// ---- DUTs/IO/PDOs/Channel_3263D8D5.TcDUT
{attribute 'GeneratedUsingTerminal: KL8524'}
{attribute addProperty BoxType "KL8524"}
{attribute addProperty Id "StateAT %I*USINT0Auto_Manual_ChannelAT %I*BYTE0Switch_modeAT %I*BYTE0On_Off_ChannelAT %I*BYTE0CtrlAT %Q*USINT0Switch_mode_OutAT %Q*BYTE0Data_Reg_ComAT %Q*BYTE0LED_Out_greenAT %Q*BYTE0LED_Out_yellowAT %Q*BYTE0"}
{attribute addProperty CRC "845404373"}
{attribute addProperty Size "0"}
TYPE Channel_3263D8D5 :
STRUCT
	{attribute addProperty Name "State"}
	State AT %I* : USINT;
	{attribute addProperty Name "Auto_Manual_Channel"}
	Auto_Manual_Channel AT %I* : BYTE;
	{attribute addProperty Name "Switch_mode"}
	Switch_mode AT %I* : BYTE;
	{attribute addProperty Name "On_Off_Channel"}
	On_Off_Channel AT %I* : BYTE;
	{attribute addProperty Name "Ctrl"}
	Ctrl AT %Q* : USINT;
	{attribute addProperty Name "Switch_mode_Out"}
	Switch_mode_Out AT %Q* : BYTE;
	{attribute addProperty Name "Data_Reg_Com"}
	Data_Reg_Com AT %Q* : BYTE;
	{attribute addProperty Name "LED_Out_green"}
	LED_Out_green AT %Q* : BYTE;
	{attribute addProperty Name "LED_Out_yellow"}
	LED_Out_yellow AT %Q* : BYTE;
END_STRUCT
END_TYPE

// ---- DUTs/IO/PDOs/Channel_D490E973.TcDUT
{attribute 'GeneratedUsingTerminal: KL8528'}
{attribute addProperty BoxType "KL8528"}
{attribute addProperty Id "StateAT %I*USINT0Auto_Manual_ChannelAT %I*BYTE0On_Off_ChannelAT %I*BYTE0CtrlAT %Q*USINT0OutAT %Q*BYTE0Data_Reg_ComAT %Q*BYTE0LED_Out_greenAT %Q*BYTE0LED_Out_yellowAT %Q*BYTE0"}
{attribute addProperty CRC "3566266739"}
{attribute addProperty Size "0"}
TYPE Channel_D490E973 :
STRUCT
	{attribute addProperty Name "State"}
	State AT %I* : USINT;
	{attribute addProperty Name "Auto_Manual_Channel"}
	Auto_Manual_Channel AT %I* : BYTE;
	{attribute addProperty Name "On_Off_Channel"}
	On_Off_Channel AT %I* : BYTE;
	{attribute addProperty Name "Ctrl"}
	Ctrl AT %Q* : USINT;
	{attribute addProperty Name "Out"}
	Out AT %Q* : BYTE;
	{attribute addProperty Name "Data_Reg_Com"}
	Data_Reg_Com AT %Q* : BYTE;
	{attribute addProperty Name "LED_Out_green"}
	LED_Out_green AT %Q* : BYTE;
	{attribute addProperty Name "LED_Out_yellow"}
	LED_Out_yellow AT %Q* : BYTE;
END_STRUCT
END_TYPE

// ---- DUTs/IO/PDOs/KL_6576A681.TcDUT
{attribute 'GeneratedUsingTerminal: KL8610'}
{attribute addProperty BoxType "KL8610"}
{attribute addProperty Id "StateAT %I*USINT0Data_InAT %I*INT0CtrlAT %Q*USINT0Data_OutAT %Q*INT0"}
{attribute addProperty CRC "1702274689"}
{attribute addProperty Size "0"}
TYPE KL_6576A681 :
STRUCT
	{attribute addProperty Name "State"}
	State AT %I* : USINT;
	{attribute addProperty Name "Data_In"}
	Data_In AT %I* : INT;
	{attribute addProperty Name "Ctrl"}
	Ctrl AT %Q* : USINT;
	{attribute addProperty Name "Data_Out"}
	Data_Out AT %Q* : INT;
END_STRUCT
END_TYPE

// ---- DUTs/IO/PDOs/Channel_64AAC8C7.TcDUT
{attribute 'GeneratedUsingTerminal: KL9110'}
{attribute addProperty BoxType "KL9110"}
{attribute addProperty Id "PowerAT %I*BOOL0ShortCircuitAT %I*BOOL0"}
{attribute addProperty CRC "1688914119"}
{attribute addProperty Size "0"}
TYPE Channel_64AAC8C7 EXTENDS InputBase_8311D824 :
STRUCT
	{attribute addProperty Name "Power"}
	Power AT %I* : BOOL;
	{attribute addProperty Name "ShortCircuit"}
	ShortCircuit AT %I* : BOOL;
END_STRUCT
END_TYPE

// ---- DUTs/IO/PDOs/Channel_471FAA5C.TcDUT
{attribute 'GeneratedUsingTerminal: KL9191'}
{attribute addProperty BoxType "KL9191"}
{attribute addProperty Id "Contact_DI1AT %I*BOOL0Contact_DI2AT %I*BOOL0Contact_DI3AT %I*BOOL0LED_DO1AT %Q*BOOL0Relay_2kWAT %Q*BOOL0Relay_FAN1AT %Q*BOOL0Relay_FAN2AT %Q*BOOL0Relay_FAN3AT %Q*BOOL0TRIAC_Y1AT %Q*BOOL0TRIAC_Y2AT %Q*BOOL0"}
{attribute addProperty CRC "1193257564"}
{attribute addProperty Size "0"}
TYPE Channel_471FAA5C :
STRUCT
	{attribute addProperty Name "Contact_DI1"}
	Contact_DI1 AT %I* : BOOL;
	{attribute addProperty Name "Contact_DI2"}
	Contact_DI2 AT %I* : BOOL;
	{attribute addProperty Name "Contact_DI3"}
	Contact_DI3 AT %I* : BOOL;
	{attribute addProperty Name "LED_DO1"}
	LED_DO1 AT %Q* : BOOL;
	{attribute addProperty Name "Relay_2kW"}
	Relay_2kW AT %Q* : BOOL;
	{attribute addProperty Name "Relay_FAN1"}
	Relay_FAN1 AT %Q* : BOOL;
	{attribute addProperty Name "Relay_FAN2"}
	Relay_FAN2 AT %Q* : BOOL;
	{attribute addProperty Name "Relay_FAN3"}
	Relay_FAN3 AT %Q* : BOOL;
	{attribute addProperty Name "TRIAC_Y1"}
	TRIAC_Y1 AT %Q* : BOOL;
	{attribute addProperty Name "TRIAC_Y2"}
	TRIAC_Y2 AT %Q* : BOOL;
END_STRUCT
END_TYPE

// ---- DUTs/IO/PDOs/Diag_1F4F4573.TcDUT
{attribute 'GeneratedUsingTerminal: KL9505-0010'}
{attribute addProperty BoxType "KL9505-0010"}
{attribute addProperty Id "Supply_Voltage_OKAT %I*BOOL0Over_currentAT %I*BOOL0"}
{attribute addProperty CRC "525288819"}
{attribute addProperty Size "0"}
TYPE Diag_1F4F4573 EXTENDS InputBase_8311D824 :
STRUCT
	{attribute addProperty Name "Supply_Voltage_OK"}
	Supply_Voltage_OK AT %I* : BOOL;
	{attribute addProperty Name "Over_current"}
	Over_current AT %I* : BOOL;
END_STRUCT
END_TYPE

// ---- DUTs/IO/PDOs/Channel_0029832E.TcDUT
{attribute 'GeneratedUsingTerminal: KL9528'}
{attribute addProperty BoxType "KL9528"}
{attribute addProperty Id "OverloadAT %I*BOOL0UndervoltageAT %I*BOOL0ResetAT %Q*BOOL0"}
{attribute addProperty CRC "2720558"}
{attribute addProperty Size "0"}
TYPE Channel_0029832E :
STRUCT
	{attribute addProperty Name "Overload"}
	Overload AT %I* : BOOL;
	{attribute addProperty Name "Undervoltage"}
	Undervoltage AT %I* : BOOL;
	{attribute addProperty Name "Reset"}
	Reset AT %Q* : BOOL;
END_STRUCT
END_TYPE

// ---- DUTs/IO/PDOs/Channel_12652743.TcDUT
{attribute 'GeneratedUsingTerminal: KL9999'}
{attribute addProperty BoxType "KL9999"}
{attribute addProperty Id "VarInAT %I*UINT0VarOutAT %Q*UINT0"}
{attribute addProperty CRC "308619075"}
{attribute addProperty Size "0"}
TYPE Channel_12652743 :
STRUCT
	{attribute addProperty Name "VarIn"}
	VarIn AT %I* : UINT;
	{attribute addProperty Name "VarOut"}
	VarOut AT %Q* : UINT;
END_STRUCT
END_TYPE

// ---- DUTs/IO/PDOs/InfoData_E68C61CD.TcDUT
{attribute 'GeneratedUsingTerminal: IODEVICETYPE_ETHERCATPROT'}
{attribute addProperty BoxType "IODEVICETYPE_ETHERCATPROT"}
{attribute addProperty Id "ChangeCountAT %I*UINT2DevIdAT %I*UINT2AmsNetIdAT %I*AMSNETID6CfgSlaveCountAT %I*UINT2DcToTcTimeOffsetAT %I*LINT8DcToExtTimeOffsetAT %I*LINT8"}
{attribute addProperty CRC "3867959757"}
{attribute addProperty Size "28"}
TYPE InfoData_E68C61CD EXTENDS InputBase_8311D824 :
STRUCT
	{attribute addProperty Name "ChangeCount"}
	ChangeCount AT %I* : UINT;
	{attribute addProperty Name "DevId"}
	DevId AT %I* : UINT;
	{attribute addProperty Name "AmsNetId"}
	AmsNetId AT %I* : AMSNETID;
	{attribute addProperty Name "CfgSlaveCount"}
	CfgSlaveCount AT %I* : UINT;
	{attribute addProperty Name "DcToTcTimeOffset"}
	DcToTcTimeOffset AT %I* : LINT;
	{attribute addProperty Name "DcToExtTimeOffset"}
	DcToExtTimeOffset AT %I* : LINT;
END_STRUCT
END_TYPE

// ---- DUTs/IO/PDOs/WcState_0B2B16F9.TcDUT
{attribute 'GeneratedUsingTerminal: IODEVICETYPE_ETHERCATPROT'}
{attribute addProperty BoxType "IODEVICETYPE_ETHERCATPROT"}
{attribute addProperty Id "WcStateAT %I*BOOL1"}
{attribute addProperty CRC "187373305"}
{attribute addProperty Size "1"}
TYPE WcState_0B2B16F9 :
STRUCT
	{attribute addProperty Name "WcState"}
	WcState AT %I* : BOOL;
END_STRUCT
END_TYPE

// ---- DUTs/IO/PDOs/InfoData_2A97D6CF.TcDUT
{attribute 'GeneratedUsingTerminal: IODEVICETYPE_ETHERCATPROT'}
{attribute addProperty BoxType "IODEVICETYPE_ETHERCATPROT"}
{attribute addProperty Id "ObjectIdAT %I*OTCID4StateAT %I*UINT2SlaveCountAT %I*UINT2"}
{attribute addProperty CRC "714593999"}
{attribute addProperty Size "8"}
TYPE InfoData_2A97D6CF EXTENDS InputBase_8311D824 :
STRUCT
	{attribute addProperty Name "ObjectId"}
	ObjectId AT %I* : OTCID;
	{attribute addProperty Name "State"}
	State AT %I* : UINT;
	{attribute addProperty Name "SlaveCount"}
	SlaveCount AT %I* : UINT;
END_STRUCT
END_TYPE

// ---- DUTs/IO/PDOs/Inputs_25A0042B.TcDUT
{attribute 'GeneratedUsingTerminal: IODEVICETYPE_ETHERCATPROT'}
{attribute addProperty BoxType "IODEVICETYPE_ETHERCATPROT"}
{attribute addProperty Id "SlaveCountAT %I*UINT2DevStateAT %I*UINT2Frm0StateAT %I*UINT2Frm0WcStateAT %I*UINT2Frm0InputToggleAT %I*UINT2Frm1StateAT %I*UINT2Frm1WcStateAT %I*UINT2Frm1InputToggleAT %I*UINT2Frm2StateAT %I*UINT2Frm2WcStateAT %I*UINT2Frm2InputToggleAT %I*UINT2Frm3StateAT %I*UINT2Frm3WcStateAT %I*UINT2Frm3InputToggleAT %I*UINT2Frm4StateAT %I*UINT2Frm4WcStateAT %I*UINT2Frm4InputToggleAT %I*UINT2Frm5StateAT %I*UINT2Frm5WcStateAT %I*UINT2Frm5InputToggleAT %I*UINT2Frm6StateAT %I*UINT2Frm6WcStateAT %I*UINT2Frm6InputToggleAT %I*UINT2Frm7StateAT %I*UINT2Frm7WcStateAT %I*UINT2Frm7InputToggleAT %I*UINT2Frm8StateAT %I*UINT2Frm8WcStateAT %I*UINT2Frm8InputToggleAT %I*UINT2Frm9StateAT %I*UINT2Frm9WcStateAT %I*UINT2Frm9InputToggleAT %I*UINT2Frm10StateAT %I*UINT2Frm10WcStateAT %I*UINT2Frm10InputToggleAT %I*UINT2Frm11StateAT %I*UINT2Frm11WcStateAT %I*UINT2Frm11InputToggleAT %I*UINT2Frm12StateAT %I*UINT2Frm12WcStateAT %I*UINT2Frm12InputToggleAT %I*UINT2Frm13StateAT %I*UINT2Frm13WcStateAT %I*UINT2Frm13InputToggleAT %I*UINT2Frm14StateAT %I*UINT2Frm14WcStateAT %I*UINT2Frm14InputToggleAT %I*UINT2Frm15StateAT %I*UINT2Frm15WcStateAT %I*UINT2Frm15InputToggleAT %I*UINT2Frm16StateAT %I*UINT2Frm16WcStateAT %I*UINT2Frm16InputToggleAT %I*UINT2Frm17StateAT %I*UINT2Frm17WcStateAT %I*UINT2Frm17InputToggleAT %I*UINT2Frm18StateAT %I*UINT2Frm18WcStateAT %I*UINT2Frm18InputToggleAT %I*UINT2Frm19StateAT %I*UINT2Frm19WcStateAT %I*UINT2Frm19InputToggleAT %I*UINT2Frm20StateAT %I*UINT2Frm20WcStateAT %I*UINT2Frm20InputToggleAT %I*UINT2Frm21StateAT %I*UINT2Frm21WcStateAT %I*UINT2Frm21InputToggleAT %I*UINT2Frm22StateAT %I*UINT2Frm22WcStateAT %I*UINT2Frm22InputToggleAT %I*UINT2Frm23StateAT %I*UINT2Frm23WcStateAT %I*UINT2Frm23InputToggleAT %I*UINT2Frm24StateAT %I*UINT2Frm24WcStateAT %I*UINT2Frm24InputToggleAT %I*UINT2Frm25StateAT %I*UINT2Frm25WcStateAT %I*UINT2Frm25InputToggleAT %I*UINT2"}
{attribute addProperty CRC "631243819"}
{attribute addProperty Size "160"}
TYPE Inputs_25A0042B EXTENDS InputBase_8311D824 :
STRUCT
	{attribute addProperty Name "SlaveCount"}
	SlaveCount AT %I* : UINT;
	{attribute addProperty Name "DevState"}
	DevState AT %I* : UINT;
	{attribute addProperty Name "Frm0State"}
	Frm0State AT %I* : UINT;
	{attribute addProperty Name "Frm0WcState"}
	Frm0WcState AT %I* : UINT;
	{attribute addProperty Name "Frm0InputToggle"}
	Frm0InputToggle AT %I* : UINT;
	{attribute addProperty Name "Frm1State"}
	Frm1State AT %I* : UINT;
	{attribute addProperty Name "Frm1WcState"}
	Frm1WcState AT %I* : UINT;
	{attribute addProperty Name "Frm1InputToggle"}
	Frm1InputToggle AT %I* : UINT;
	{attribute addProperty Name "Frm2State"}
	Frm2State AT %I* : UINT;
	{attribute addProperty Name "Frm2WcState"}
	Frm2WcState AT %I* : UINT;
	{attribute addProperty Name "Frm2InputToggle"}
	Frm2InputToggle AT %I* : UINT;
	{attribute addProperty Name "Frm3State"}
	Frm3State AT %I* : UINT;
	{attribute addProperty Name "Frm3WcState"}
	Frm3WcState AT %I* : UINT;
	{attribute addProperty Name "Frm3InputToggle"}
	Frm3InputToggle AT %I* : UINT;
	{attribute addProperty Name "Frm4State"}
	Frm4State AT %I* : UINT;
	{attribute addProperty Name "Frm4WcState"}
	Frm4WcState AT %I* : UINT;
	{attribute addProperty Name "Frm4InputToggle"}
	Frm4InputToggle AT %I* : UINT;
	{attribute addProperty Name "Frm5State"}
	Frm5State AT %I* : UINT;
	{attribute addProperty Name "Frm5WcState"}
	Frm5WcState AT %I* : UINT;
	{attribute addProperty Name "Frm5InputToggle"}
	Frm5InputToggle AT %I* : UINT;
	{attribute addProperty Name "Frm6State"}
	Frm6State AT %I* : UINT;
	{attribute addProperty Name "Frm6WcState"}
	Frm6WcState AT %I* : UINT;
	{attribute addProperty Name "Frm6InputToggle"}
	Frm6InputToggle AT %I* : UINT;
	{attribute addProperty Name "Frm7State"}
	Frm7State AT %I* : UINT;
	{attribute addProperty Name "Frm7WcState"}
	Frm7WcState AT %I* : UINT;
	{attribute addProperty Name "Frm7InputToggle"}
	Frm7InputToggle AT %I* : UINT;
	{attribute addProperty Name "Frm8State"}
	Frm8State AT %I* : UINT;
	{attribute addProperty Name "Frm8WcState"}
	Frm8WcState AT %I* : UINT;
	{attribute addProperty Name "Frm8InputToggle"}
	Frm8InputToggle AT %I* : UINT;
	{attribute addProperty Name "Frm9State"}
	Frm9State AT %I* : UINT;
	{attribute addProperty Name "Frm9WcState"}
	Frm9WcState AT %I* : UINT;
	{attribute addProperty Name "Frm9InputToggle"}
	Frm9InputToggle AT %I* : UINT;
	{attribute addProperty Name "Frm10State"}
	Frm10State AT %I* : UINT;
	{attribute addProperty Name "Frm10WcState"}
	Frm10WcState AT %I* : UINT;
	{attribute addProperty Name "Frm10InputToggle"}
	Frm10InputToggle AT %I* : UINT;
	{attribute addProperty Name "Frm11State"}
	Frm11State AT %I* : UINT;
	{attribute addProperty Name "Frm11WcState"}
	Frm11WcState AT %I* : UINT;
	{attribute addProperty Name "Frm11InputToggle"}
	Frm11InputToggle AT %I* : UINT;
	{attribute addProperty Name "Frm12State"}
	Frm12State AT %I* : UINT;
	{attribute addProperty Name "Frm12WcState"}
	Frm12WcState AT %I* : UINT;
	{attribute addProperty Name "Frm12InputToggle"}
	Frm12InputToggle AT %I* : UINT;
	{attribute addProperty Name "Frm13State"}
	Frm13State AT %I* : UINT;
	{attribute addProperty Name "Frm13WcState"}
	Frm13WcState AT %I* : UINT;
	{attribute addProperty Name "Frm13InputToggle"}
	Frm13InputToggle AT %I* : UINT;
	{attribute addProperty Name "Frm14State"}
	Frm14State AT %I* : UINT;
	{attribute addProperty Name "Frm14WcState"}
	Frm14WcState AT %I* : UINT;
	{attribute addProperty Name "Frm14InputToggle"}
	Frm14InputToggle AT %I* : UINT;
	{attribute addProperty Name "Frm15State"}
	Frm15State AT %I* : UINT;
	{attribute addProperty Name "Frm15WcState"}
	Frm15WcState AT %I* : UINT;
	{attribute addProperty Name "Frm15InputToggle"}
	Frm15InputToggle AT %I* : UINT;
	{attribute addProperty Name "Frm16State"}
	Frm16State AT %I* : UINT;
	{attribute addProperty Name "Frm16WcState"}
	Frm16WcState AT %I* : UINT;
	{attribute addProperty Name "Frm16InputToggle"}
	Frm16InputToggle AT %I* : UINT;
	{attribute addProperty Name "Frm17State"}
	Frm17State AT %I* : UINT;
	{attribute addProperty Name "Frm17WcState"}
	Frm17WcState AT %I* : UINT;
	{attribute addProperty Name "Frm17InputToggle"}
	Frm17InputToggle AT %I* : UINT;
	{attribute addProperty Name "Frm18State"}
	Frm18State AT %I* : UINT;
	{attribute addProperty Name "Frm18WcState"}
	Frm18WcState AT %I* : UINT;
	{attribute addProperty Name "Frm18InputToggle"}
	Frm18InputToggle AT %I* : UINT;
	{attribute addProperty Name "Frm19State"}
	Frm19State AT %I* : UINT;
	{attribute addProperty Name "Frm19WcState"}
	Frm19WcState AT %I* : UINT;
	{attribute addProperty Name "Frm19InputToggle"}
	Frm19InputToggle AT %I* : UINT;
	{attribute addProperty Name "Frm20State"}
	Frm20State AT %I* : UINT;
	{attribute addProperty Name "Frm20WcState"}
	Frm20WcState AT %I* : UINT;
	{attribute addProperty Name "Frm20InputToggle"}
	Frm20InputToggle AT %I* : UINT;
	{attribute addProperty Name "Frm21State"}
	Frm21State AT %I* : UINT;
	{attribute addProperty Name "Frm21WcState"}
	Frm21WcState AT %I* : UINT;
	{attribute addProperty Name "Frm21InputToggle"}
	Frm21InputToggle AT %I* : UINT;
	{attribute addProperty Name "Frm22State"}
	Frm22State AT %I* : UINT;
	{attribute addProperty Name "Frm22WcState"}
	Frm22WcState AT %I* : UINT;
	{attribute addProperty Name "Frm22InputToggle"}
	Frm22InputToggle AT %I* : UINT;
	{attribute addProperty Name "Frm23State"}
	Frm23State AT %I* : UINT;
	{attribute addProperty Name "Frm23WcState"}
	Frm23WcState AT %I* : UINT;
	{attribute addProperty Name "Frm23InputToggle"}
	Frm23InputToggle AT %I* : UINT;
	{attribute addProperty Name "Frm24State"}
	Frm24State AT %I* : UINT;
	{attribute addProperty Name "Frm24WcState"}
	Frm24WcState AT %I* : UINT;
	{attribute addProperty Name "Frm24InputToggle"}
	Frm24InputToggle AT %I* : UINT;
	{attribute addProperty Name "Frm25State"}
	Frm25State AT %I* : UINT;
	{attribute addProperty Name "Frm25WcState"}
	Frm25WcState AT %I* : UINT;
	{attribute addProperty Name "Frm25InputToggle"}
	Frm25InputToggle AT %I* : UINT;
END_STRUCT
END_TYPE

// ---- DUTs/IO/PDOs/Outputs_2397A10E.TcDUT
{attribute 'GeneratedUsingTerminal: IODEVICETYPE_ETHERCATPROT'}
{attribute addProperty BoxType "IODEVICETYPE_ETHERCATPROT"}
{attribute addProperty Id "DevCtrlAT %Q*UINT2Frm0CtrlAT %Q*UINT2Frm0WcCtrlAT %Q*UINT2Frm1CtrlAT %Q*UINT2Frm1WcCtrlAT %Q*UINT2Frm2CtrlAT %Q*UINT2Frm2WcCtrlAT %Q*UINT2Frm3CtrlAT %Q*UINT2Frm3WcCtrlAT %Q*UINT2Frm4CtrlAT %Q*UINT2Frm4WcCtrlAT %Q*UINT2Frm5CtrlAT %Q*UINT2Frm5WcCtrlAT %Q*UINT2Frm6CtrlAT %Q*UINT2Frm6WcCtrlAT %Q*UINT2Frm7CtrlAT %Q*UINT2Frm7WcCtrlAT %Q*UINT2Frm8CtrlAT %Q*UINT2Frm8WcCtrlAT %Q*UINT2Frm9CtrlAT %Q*UINT2Frm9WcCtrlAT %Q*UINT2Frm10CtrlAT %Q*UINT2Frm10WcCtrlAT %Q*UINT2Frm11CtrlAT %Q*UINT2Frm11WcCtrlAT %Q*UINT2Frm12CtrlAT %Q*UINT2Frm12WcCtrlAT %Q*UINT2Frm13CtrlAT %Q*UINT2Frm13WcCtrlAT %Q*UINT2Frm14CtrlAT %Q*UINT2Frm14WcCtrlAT %Q*UINT2Frm15CtrlAT %Q*UINT2Frm15WcCtrlAT %Q*UINT2Frm16CtrlAT %Q*UINT2Frm16WcCtrlAT %Q*UINT2Frm17CtrlAT %Q*UINT2Frm17WcCtrlAT %Q*UINT2Frm18CtrlAT %Q*UINT2Frm18WcCtrlAT %Q*UINT2Frm19CtrlAT %Q*UINT2Frm19WcCtrlAT %Q*UINT2Frm20CtrlAT %Q*UINT2Frm20WcCtrlAT %Q*UINT2Frm21CtrlAT %Q*UINT2Frm21WcCtrlAT %Q*UINT2Frm22CtrlAT %Q*UINT2Frm22WcCtrlAT %Q*UINT2Frm23CtrlAT %Q*UINT2Frm23WcCtrlAT %Q*UINT2Frm24CtrlAT %Q*UINT2Frm24WcCtrlAT %Q*UINT2Frm25CtrlAT %Q*UINT2Frm25WcCtrlAT %Q*UINT2"}
{attribute addProperty CRC "597139726"}
{attribute addProperty Size "106"}
TYPE Outputs_2397A10E EXTENDS OutputBase_10CEE7DE :
STRUCT
	{attribute addProperty Name "DevCtrl"}
	DevCtrl AT %Q* : UINT;
	{attribute addProperty Name "Frm0Ctrl"}
	Frm0Ctrl AT %Q* : UINT;
	{attribute addProperty Name "Frm0WcCtrl"}
	Frm0WcCtrl AT %Q* : UINT;
	{attribute addProperty Name "Frm1Ctrl"}
	Frm1Ctrl AT %Q* : UINT;
	{attribute addProperty Name "Frm1WcCtrl"}
	Frm1WcCtrl AT %Q* : UINT;
	{attribute addProperty Name "Frm2Ctrl"}
	Frm2Ctrl AT %Q* : UINT;
	{attribute addProperty Name "Frm2WcCtrl"}
	Frm2WcCtrl AT %Q* : UINT;
	{attribute addProperty Name "Frm3Ctrl"}
	Frm3Ctrl AT %Q* : UINT;
	{attribute addProperty Name "Frm3WcCtrl"}
	Frm3WcCtrl AT %Q* : UINT;
	{attribute addProperty Name "Frm4Ctrl"}
	Frm4Ctrl AT %Q* : UINT;
	{attribute addProperty Name "Frm4WcCtrl"}
	Frm4WcCtrl AT %Q* : UINT;
	{attribute addProperty Name "Frm5Ctrl"}
	Frm5Ctrl AT %Q* : UINT;
	{attribute addProperty Name "Frm5WcCtrl"}
	Frm5WcCtrl AT %Q* : UINT;
	{attribute addProperty Name "Frm6Ctrl"}
	Frm6Ctrl AT %Q* : UINT;
	{attribute addProperty Name "Frm6WcCtrl"}
	Frm6WcCtrl AT %Q* : UINT;
	{attribute addProperty Name "Frm7Ctrl"}
	Frm7Ctrl AT %Q* : UINT;
	{attribute addProperty Name "Frm7WcCtrl"}
	Frm7WcCtrl AT %Q* : UINT;
	{attribute addProperty Name "Frm8Ctrl"}
	Frm8Ctrl AT %Q* : UINT;
	{attribute addProperty Name "Frm8WcCtrl"}
	Frm8WcCtrl AT %Q* : UINT;
	{attribute addProperty Name "Frm9Ctrl"}
	Frm9Ctrl AT %Q* : UINT;
	{attribute addProperty Name "Frm9WcCtrl"}
	Frm9WcCtrl AT %Q* : UINT;
	{attribute addProperty Name "Frm10Ctrl"}
	Frm10Ctrl AT %Q* : UINT;
	{attribute addProperty Name "Frm10WcCtrl"}
	Frm10WcCtrl AT %Q* : UINT;
	{attribute addProperty Name "Frm11Ctrl"}
	Frm11Ctrl AT %Q* : UINT;
	{attribute addProperty Name "Frm11WcCtrl"}
	Frm11WcCtrl AT %Q* : UINT;
	{attribute addProperty Name "Frm12Ctrl"}
	Frm12Ctrl AT %Q* : UINT;
	{attribute addProperty Name "Frm12WcCtrl"}
	Frm12WcCtrl AT %Q* : UINT;
	{attribute addProperty Name "Frm13Ctrl"}
	Frm13Ctrl AT %Q* : UINT;
	{attribute addProperty Name "Frm13WcCtrl"}
	Frm13WcCtrl AT %Q* : UINT;
	{attribute addProperty Name "Frm14Ctrl"}
	Frm14Ctrl AT %Q* : UINT;
	{attribute addProperty Name "Frm14WcCtrl"}
	Frm14WcCtrl AT %Q* : UINT;
	{attribute addProperty Name "Frm15Ctrl"}
	Frm15Ctrl AT %Q* : UINT;
	{attribute addProperty Name "Frm15WcCtrl"}
	Frm15WcCtrl AT %Q* : UINT;
	{attribute addProperty Name "Frm16Ctrl"}
	Frm16Ctrl AT %Q* : UINT;
	{attribute addProperty Name "Frm16WcCtrl"}
	Frm16WcCtrl AT %Q* : UINT;
	{attribute addProperty Name "Frm17Ctrl"}
	Frm17Ctrl AT %Q* : UINT;
	{attribute addProperty Name "Frm17WcCtrl"}
	Frm17WcCtrl AT %Q* : UINT;
	{attribute addProperty Name "Frm18Ctrl"}
	Frm18Ctrl AT %Q* : UINT;
	{attribute addProperty Name "Frm18WcCtrl"}
	Frm18WcCtrl AT %Q* : UINT;
	{attribute addProperty Name "Frm19Ctrl"}
	Frm19Ctrl AT %Q* : UINT;
	{attribute addProperty Name "Frm19WcCtrl"}
	Frm19WcCtrl AT %Q* : UINT;
	{attribute addProperty Name "Frm20Ctrl"}
	Frm20Ctrl AT %Q* : UINT;
	{attribute addProperty Name "Frm20WcCtrl"}
	Frm20WcCtrl AT %Q* : UINT;
	{attribute addProperty Name "Frm21Ctrl"}
	Frm21Ctrl AT %Q* : UINT;
	{attribute addProperty Name "Frm21WcCtrl"}
	Frm21WcCtrl AT %Q* : UINT;
	{attribute addProperty Name "Frm22Ctrl"}
	Frm22Ctrl AT %Q* : UINT;
	{attribute addProperty Name "Frm22WcCtrl"}
	Frm22WcCtrl AT %Q* : UINT;
	{attribute addProperty Name "Frm23Ctrl"}
	Frm23Ctrl AT %Q* : UINT;
	{attribute addProperty Name "Frm23WcCtrl"}
	Frm23WcCtrl AT %Q* : UINT;
	{attribute addProperty Name "Frm24Ctrl"}
	Frm24Ctrl AT %Q* : UINT;
	{attribute addProperty Name "Frm24WcCtrl"}
	Frm24WcCtrl AT %Q* : UINT;
	{attribute addProperty Name "Frm25Ctrl"}
	Frm25Ctrl AT %Q* : UINT;
	{attribute addProperty Name "Frm25WcCtrl"}
	Frm25WcCtrl AT %Q* : UINT;
END_STRUCT
END_TYPE

// ---- DUTs/IO/Boxes/EK1100_1FC0878B.TcDUT
{attribute 'GeneratedUsingTerminal: EK1100-0000-0018'}
{attribute addProperty BoxType "EK1100-0000-0018"}
{attribute addProperty Description "EK1100 EtherCAT Coupler (2A E-Bus)"}
{attribute addProperty Physics "YKY"}
{attribute addProperty Id "InfoDataAT %I*InfoData_6F19DB2B2"}
{attribute addProperty CRC "532711307"}
{attribute addProperty Size "2"}
TYPE EK1100_1FC0878B EXTENDS EtcSlaveBoxBase_77A0E4A7 :
STRUCT
	{attribute addProperty Name "InfoData"}
	InfoData : InfoData_6F19DB2B;
END_STRUCT
END_TYPE

// ---- DUTs/IO/Boxes/EK1122_1FC0878B.TcDUT
{attribute 'GeneratedUsingTerminal: EK1122-0000-0018'}
{attribute addProperty BoxType "EK1122-0000-0018"}
{attribute addProperty Description "EK1122 2 port EtherCAT junction"}
{attribute addProperty Physics "KYKY"}
{attribute addProperty Id "InfoDataAT %I*InfoData_6F19DB2B2"}
{attribute addProperty CRC "532711307"}
{attribute addProperty Size "2"}
TYPE EK1122_1FC0878B EXTENDS EtcSlaveTerminalBase_947E5A46 :
STRUCT
	{attribute addProperty Name "InfoData"}
	InfoData : InfoData_6F19DB2B;
END_STRUCT
END_TYPE

// ---- DUTs/IO/Boxes/BK1250_A2FCADE7.TcDUT
{attribute 'GeneratedUsingTerminal: BK1250-0000-0000'}
{attribute addProperty BoxType "BK1250-0000-0000"}
{attribute addProperty Description ""}
{attribute addProperty Physics "K"}
{attribute addProperty Id "InputsAT %I*Inputs_CC16D1F40OutputsAT %I*Outputs_D8BAB3B30WcStateAT %I*WcState_9091E0EB2InfoDataAT %I*InfoData_90184F0C16"}
{attribute addProperty CRC "2734468583"}
{attribute addProperty Size "18"}
TYPE BK1250_A2FCADE7 EXTENDS EtcSlaveTerminalBase_947E5A46 :
STRUCT
	{attribute addProperty Name "Inputs"}
	Inputs : Inputs_CC16D1F4;
	{attribute addProperty Name "Outputs"}
	Outputs : Outputs_D8BAB3B3;
	{attribute addProperty Name "WcState"}
	WcState : WcState_9091E0EB;
	{attribute addProperty Name "InfoData"}
	InfoData : InfoData_90184F0C;
END_STRUCT
END_TYPE

// ---- DUTs/IO/Boxes/KL1002_BB38DA8F.TcDUT
{attribute 'GeneratedUsingTerminal: KL1002'}
{attribute addProperty BoxType "KL1002"}
{attribute addProperty Description ""}
{attribute addProperty Physics ""}
{attribute addProperty Id "Channel_1AT %I*Channel_87C95E760Channel_2AT %I*Channel_87C95E760"}
{attribute addProperty CRC "3141065359"}
{attribute addProperty Size "0"}
TYPE KL1002_BB38DA8F :
STRUCT
	{attribute addProperty Name "Channel_1"}
	Channel_1 : Channel_87C95E76;
	{attribute addProperty Name "Channel_2"}
	Channel_2 : Channel_87C95E76;
END_STRUCT
END_TYPE

// ---- DUTs/IO/Boxes/BK1120_6D44499E.TcDUT
{attribute 'GeneratedUsingTerminal: BK1120-0000-0000'}
{attribute addProperty BoxType "BK1120-0000-0000"}
{attribute addProperty Description ""}
{attribute addProperty Physics "YY"}
{attribute addProperty Id "InputsAT %I*Inputs_CC16D1F40OutputsAT %I*Outputs_D8BAB3B30WcStateAT %I*WcState_9091E0EB2InfoDataAT %I*InfoData_32EB74EA10"}
{attribute addProperty CRC "1833191838"}
{attribute addProperty Size "12"}
TYPE BK1120_6D44499E EXTENDS EtcSlaveBoxBase_77A0E4A7 :
STRUCT
	{attribute addProperty Name "Inputs"}
	Inputs : Inputs_CC16D1F4;
	{attribute addProperty Name "Outputs"}
	Outputs : Outputs_D8BAB3B3;
	{attribute addProperty Name "WcState"}
	WcState : WcState_9091E0EB;
	{attribute addProperty Name "InfoData"}
	InfoData : InfoData_32EB74EA;
END_STRUCT
END_TYPE

// ---- DUTs/IO/Boxes/BK1120_A2FCADE7.TcDUT
{attribute 'GeneratedUsingTerminal: BK1120-0000-0001'}
{attribute addProperty BoxType "BK1120-0000-0001"}
{attribute addProperty Description ""}
{attribute addProperty Physics "YY"}
{attribute addProperty Id "InputsAT %I*Inputs_CC16D1F40OutputsAT %I*Outputs_D8BAB3B30WcStateAT %I*WcState_9091E0EB2InfoDataAT %I*InfoData_90184F0C16"}
{attribute addProperty CRC "2734468583"}
{attribute addProperty Size "18"}
TYPE BK1120_A2FCADE7 EXTENDS EtcSlaveBoxBase_77A0E4A7 :
STRUCT
	{attribute addProperty Name "Inputs"}
	Inputs : Inputs_CC16D1F4;
	{attribute addProperty Name "Outputs"}
	Outputs : Outputs_D8BAB3B3;
	{attribute addProperty Name "WcState"}
	WcState : WcState_9091E0EB;
	{attribute addProperty Name "InfoData"}
	InfoData : InfoData_90184F0C;
END_STRUCT
END_TYPE

// ---- DUTs/IO/Boxes/CPXXXX_A2FCADE7.TcDUT
{attribute 'GeneratedUsingTerminal: CPXXXX-BK7902-0016'}
{attribute addProperty BoxType "CPXXXX-BK7902-0016"}
{attribute addProperty Description ""}
{attribute addProperty Physics "YY"}
{attribute addProperty Id "InputsAT %I*Inputs_CC16D1F40OutputsAT %I*Outputs_D8BAB3B30WcStateAT %I*WcState_9091E0EB2InfoDataAT %I*InfoData_90184F0C16"}
{attribute addProperty CRC "2734468583"}
{attribute addProperty Size "18"}
TYPE CPXXXX_A2FCADE7 EXTENDS EtcSlaveBoxBase_77A0E4A7 :
STRUCT
	{attribute addProperty Name "Inputs"}
	Inputs : Inputs_CC16D1F4;
	{attribute addProperty Name "Outputs"}
	Outputs : Outputs_D8BAB3B3;
	{attribute addProperty Name "WcState"}
	WcState : WcState_9091E0EB;
	{attribute addProperty Name "InfoData"}
	InfoData : InfoData_90184F0C;
END_STRUCT
END_TYPE

// ---- DUTs/IO/Boxes/BK1150_A2FCADE7.TcDUT
{attribute 'GeneratedUsingTerminal: BK1150-0000-0016'}
{attribute addProperty BoxType "BK1150-0000-0016"}
{attribute addProperty Description ""}
{attribute addProperty Physics "YY"}
{attribute addProperty Id "InputsAT %I*Inputs_CC16D1F40OutputsAT %I*Outputs_D8BAB3B30WcStateAT %I*WcState_9091E0EB2InfoDataAT %I*InfoData_90184F0C16"}
{attribute addProperty CRC "2734468583"}
{attribute addProperty Size "18"}
TYPE BK1150_A2FCADE7 EXTENDS EtcSlaveBoxBase_77A0E4A7 :
STRUCT
	{attribute addProperty Name "Inputs"}
	Inputs : Inputs_CC16D1F4;
	{attribute addProperty Name "Outputs"}
	Outputs : Outputs_D8BAB3B3;
	{attribute addProperty Name "WcState"}
	WcState : WcState_9091E0EB;
	{attribute addProperty Name "InfoData"}
	InfoData : InfoData_90184F0C;
END_STRUCT
END_TYPE

// ---- DUTs/IO/Boxes/IL2300_A2FCADE7.TcDUT
{attribute 'GeneratedUsingTerminal: IL2300-B110-0016'}
{attribute addProperty BoxType "IL2300-B110-0016"}
{attribute addProperty Description ""}
{attribute addProperty Physics "YY"}
{attribute addProperty Id "InputsAT %I*Inputs_CC16D1F40OutputsAT %I*Outputs_D8BAB3B30WcStateAT %I*WcState_9091E0EB2InfoDataAT %I*InfoData_90184F0C16"}
{attribute addProperty CRC "2734468583"}
{attribute addProperty Size "18"}
TYPE IL2300_A2FCADE7 EXTENDS EtcSlaveBoxBase_77A0E4A7 :
STRUCT
	{attribute addProperty Name "Inputs"}
	Inputs : Inputs_CC16D1F4;
	{attribute addProperty Name "Outputs"}
	Outputs : Outputs_D8BAB3B3;
	{attribute addProperty Name "WcState"}
	WcState : WcState_9091E0EB;
	{attribute addProperty Name "InfoData"}
	InfoData : InfoData_90184F0C;
END_STRUCT
END_TYPE

// ---- DUTs/IO/Boxes/KL_D4CFBC22.TcDUT
{attribute 'GeneratedUsingTerminal: KL2300-0100'}
{attribute addProperty BoxType "KL2300-0100"}
{attribute addProperty Description ""}
{attribute addProperty Physics ""}
{attribute addProperty Id "Channel_1AT %Q*Channel_70C997F30Channel_2AT %Q*Channel_70C997F30Channel_3AT %Q*Channel_70C997F30Channel_4AT %Q*Channel_70C997F30"}
{attribute addProperty CRC "3570383906"}
{attribute addProperty Size "0"}
TYPE KL_D4CFBC22 :
STRUCT
	{attribute addProperty Name "Channel_1"}
	Channel_1 : Channel_70C997F3;
	{attribute addProperty Name "Channel_2"}
	Channel_2 : Channel_70C997F3;
	{attribute addProperty Name "Channel_3"}
	Channel_3 : Channel_70C997F3;
	{attribute addProperty Name "Channel_4"}
	Channel_4 : Channel_70C997F3;
END_STRUCT
END_TYPE

// ---- DUTs/IO/Boxes/KL_8EF4D3E9.TcDUT
{attribute 'GeneratedUsingTerminal: KL1000-0100'}
{attribute addProperty BoxType "KL1000-0100"}
{attribute addProperty Description ""}
{attribute addProperty Physics ""}
{attribute addProperty Id "Channel_1AT %I*Channel_87C95E760Channel_2AT %I*Channel_87C95E760Channel_3AT %I*Channel_87C95E760Channel_4AT %I*Channel_87C95E760Channel_5AT %I*Channel_87C95E760Channel_6AT %I*Channel_87C95E760Channel_7AT %I*Channel_87C95E760Channel_8AT %I*Channel_87C95E760"}
{attribute addProperty CRC "2398409705"}
{attribute addProperty Size "0"}
TYPE KL_8EF4D3E9 :
STRUCT
	{attribute addProperty Name "Channel_1"}
	Channel_1 : Channel_87C95E76;
	{attribute addProperty Name "Channel_2"}
	Channel_2 : Channel_87C95E76;
	{attribute addProperty Name "Channel_3"}
	Channel_3 : Channel_87C95E76;
	{attribute addProperty Name "Channel_4"}
	Channel_4 : Channel_87C95E76;
	{attribute addProperty Name "Channel_5"}
	Channel_5 : Channel_87C95E76;
	{attribute addProperty Name "Channel_6"}
	Channel_6 : Channel_87C95E76;
	{attribute addProperty Name "Channel_7"}
	Channel_7 : Channel_87C95E76;
	{attribute addProperty Name "Channel_8"}
	Channel_8 : Channel_87C95E76;
END_STRUCT
END_TYPE

// ---- DUTs/IO/Boxes/IL2301_A2FCADE7.TcDUT
{attribute 'GeneratedUsingTerminal: IL2301-B110-0016'}
{attribute addProperty BoxType "IL2301-B110-0016"}
{attribute addProperty Description ""}
{attribute addProperty Physics "YY"}
{attribute addProperty Id "InputsAT %I*Inputs_CC16D1F40OutputsAT %I*Outputs_D8BAB3B30WcStateAT %I*WcState_9091E0EB2InfoDataAT %I*InfoData_90184F0C16"}
{attribute addProperty CRC "2734468583"}
{attribute addProperty Size "18"}
TYPE IL2301_A2FCADE7 EXTENDS EtcSlaveBoxBase_77A0E4A7 :
STRUCT
	{attribute addProperty Name "Inputs"}
	Inputs : Inputs_CC16D1F4;
	{attribute addProperty Name "Outputs"}
	Outputs : Outputs_D8BAB3B3;
	{attribute addProperty Name "WcState"}
	WcState : WcState_9091E0EB;
	{attribute addProperty Name "InfoData"}
	InfoData : InfoData_90184F0C;
END_STRUCT
END_TYPE

// ---- DUTs/IO/Boxes/IL2302_A2FCADE7.TcDUT
{attribute 'GeneratedUsingTerminal: IL2302-B110-0016'}
{attribute addProperty BoxType "IL2302-B110-0016"}
{attribute addProperty Description ""}
{attribute addProperty Physics "YY"}
{attribute addProperty Id "InputsAT %I*Inputs_CC16D1F40OutputsAT %I*Outputs_D8BAB3B30WcStateAT %I*WcState_9091E0EB2InfoDataAT %I*InfoData_90184F0C16"}
{attribute addProperty CRC "2734468583"}
{attribute addProperty Size "18"}
TYPE IL2302_A2FCADE7 EXTENDS EtcSlaveBoxBase_77A0E4A7 :
STRUCT
	{attribute addProperty Name "Inputs"}
	Inputs : Inputs_CC16D1F4;
	{attribute addProperty Name "Outputs"}
	Outputs : Outputs_D8BAB3B3;
	{attribute addProperty Name "WcState"}
	WcState : WcState_9091E0EB;
	{attribute addProperty Name "InfoData"}
	InfoData : InfoData_90184F0C;
END_STRUCT
END_TYPE

// ---- DUTs/IO/Boxes/CU1123_1FC0878B.TcDUT
{attribute 'GeneratedUsingTerminal: CU1123-0000-0016'}
{attribute addProperty BoxType "CU1123-0000-0016"}
{attribute addProperty Description "CU1123 EtherCAT junction (3-ports)"}
{attribute addProperty Physics "Y_YY"}
{attribute addProperty Id "InfoDataAT %I*InfoData_6F19DB2B2"}
{attribute addProperty CRC "532711307"}
{attribute addProperty Size "2"}
TYPE CU1123_1FC0878B EXTENDS EtcSlaveBoxBase_77A0E4A7 :
STRUCT
	{attribute addProperty Name "InfoData"}
	InfoData : InfoData_6F19DB2B;
END_STRUCT
END_TYPE

// ---- DUTs/IO/Boxes/CU1124_1FC0878B.TcDUT
{attribute 'GeneratedUsingTerminal: CU1124-0000-0016'}
{attribute addProperty BoxType "CU1124-0000-0016"}
{attribute addProperty Description "CU1124 EtherCAT junction (4-ports)"}
{attribute addProperty Physics "YYYY"}
{attribute addProperty Id "InfoDataAT %I*InfoData_6F19DB2B2"}
{attribute addProperty CRC "532711307"}
{attribute addProperty Size "2"}
TYPE CU1124_1FC0878B EXTENDS EtcSlaveBoxBase_77A0E4A7 :
STRUCT
	{attribute addProperty Name "InfoData"}
	InfoData : InfoData_6F19DB2B;
END_STRUCT
END_TYPE

// ---- DUTs/IO/Boxes/CU1128_1FC0878B.TcDUT
{attribute 'GeneratedUsingTerminal: CU1128--0000'}
{attribute addProperty BoxType "CU1128--0000"}
{attribute addProperty Description "CU1128 6x EtherCAT junction"}
{attribute addProperty Physics "YYKY"}
{attribute addProperty Id "InfoDataAT %I*InfoData_6F19DB2B2"}
{attribute addProperty CRC "532711307"}
{attribute addProperty Size "2"}
TYPE CU1128_1FC0878B EXTENDS EtcSlaveBoxBase_77A0E4A7 :
STRUCT
	{attribute addProperty Name "InfoData"}
	InfoData : InfoData_6F19DB2B;
END_STRUCT
END_TYPE

// ---- DUTs/IO/Boxes/CU1521_1FC0878B.TcDUT
{attribute 'GeneratedUsingTerminal: CU1521-0010-0000'}
{attribute addProperty BoxType "CU1521-0010-0000"}
{attribute addProperty Description "CU1521-0010 EtherCAT media converter (Singlemode)"}
{attribute addProperty Physics "YY"}
{attribute addProperty Id "InfoDataAT %I*InfoData_6F19DB2B2"}
{attribute addProperty CRC "532711307"}
{attribute addProperty Size "2"}
TYPE CU1521_1FC0878B EXTENDS EtcSlaveBoxBase_77A0E4A7 :
STRUCT
	{attribute addProperty Name "InfoData"}
	InfoData : InfoData_6F19DB2B;
END_STRUCT
END_TYPE

// ---- DUTs/IO/Boxes/CU1561_1FC0878B.TcDUT
{attribute 'GeneratedUsingTerminal: CU1561--0000'}
{attribute addProperty BoxType "CU1561--0000"}
{attribute addProperty Description "CU1561 EtherCAT media converter (POF)"}
{attribute addProperty Physics "YY"}
{attribute addProperty Id "InfoDataAT %I*InfoData_6F19DB2B2"}
{attribute addProperty CRC "532711307"}
{attribute addProperty Size "2"}
TYPE CU1561_1FC0878B EXTENDS EtcSlaveBoxBase_77A0E4A7 :
STRUCT
	{attribute addProperty Name "InfoData"}
	InfoData : InfoData_6F19DB2B;
END_STRUCT
END_TYPE

// ---- DUTs/IO/Boxes/CU2508_1FC0878B.TcDUT
{attribute 'GeneratedUsingTerminal: CU2508--0000'}
{attribute addProperty BoxType "CU2508--0000"}
{attribute addProperty Description "CU2508 Ethernet Port"}
{attribute addProperty Physics "YY"}
{attribute addProperty Id "InfoDataAT %I*InfoData_6F19DB2B2"}
{attribute addProperty CRC "532711307"}
{attribute addProperty Size "2"}
TYPE CU2508_1FC0878B EXTENDS EtcSlaveBoxBase_77A0E4A7 :
STRUCT
	{attribute addProperty Name "InfoData"}
	InfoData : InfoData_6F19DB2B;
END_STRUCT
END_TYPE

// ---- DUTs/IO/Boxes/CU2508_EEB2FEF4.TcDUT
{attribute 'GeneratedUsingTerminal: CU2508-0000-0016'}
{attribute addProperty BoxType "CU2508-0000-0016"}
{attribute addProperty Description "CU2508 Configuration Port"}
{attribute addProperty Physics "YY"}
{attribute addProperty Id "InfoDataAT %I*InfoData_32EB74EA10"}
{attribute addProperty CRC "4004708084"}
{attribute addProperty Size "10"}
TYPE CU2508_EEB2FEF4 EXTENDS EtcSlaveBoxBase_77A0E4A7 :
STRUCT
	{attribute addProperty Name "InfoData"}
	InfoData : InfoData_32EB74EA;
END_STRUCT
END_TYPE

// ---- DUTs/IO/Boxes/CU2508_6BF2ACBC.TcDUT
{attribute 'GeneratedUsingTerminal: CU2508-0000-0017'}
{attribute addProperty BoxType "CU2508-0000-0017"}
{attribute addProperty Description "CU2508 Configuration Port"}
{attribute addProperty Physics "YY"}
{attribute addProperty Id "EPM_Inputs_Channel_1AT %I*EPM_Inputs_Channel_385E794A2EPM_Inputs_Channel_2AT %I*EPM_Inputs_Channel_385E794A2EPM_Inputs_Channel_3AT %I*EPM_Inputs_Channel_385E794A2EPM_Inputs_Channel_4AT %I*EPM_Inputs_Channel_385E794A2EPM_Inputs_Channel_5AT %I*EPM_Inputs_Channel_385E794A2EPM_Inputs_Channel_6AT %I*EPM_Inputs_Channel_385E794A2EPM_Inputs_Channel_7AT %I*EPM_Inputs_Channel_385E794A2EPM_Inputs_Channel_8AT %I*EPM_Inputs_Channel_385E794A2EPM_Inputs_Channel_9AT %I*EPM_Inputs_Channel_385E794A2EPM_Inputs_Channel_10AT %I*EPM_Inputs_Channel_385E794A2WcStateAT %I*WcState_9091E0EB2InfoDataAT %I*InfoData_32EB74EA10"}
{attribute addProperty CRC "1811066044"}
{attribute addProperty Size "32"}
TYPE CU2508_6BF2ACBC EXTENDS EtcSlaveBoxBase_77A0E4A7 :
STRUCT
	{attribute addProperty Name "EPM_Inputs_Channel_1"}
	EPM_Inputs_Channel_1 : EPM_Inputs_Channel_385E794A;
	{attribute addProperty Name "EPM_Inputs_Channel_2"}
	EPM_Inputs_Channel_2 : EPM_Inputs_Channel_385E794A;
	{attribute addProperty Name "EPM_Inputs_Channel_3"}
	EPM_Inputs_Channel_3 : EPM_Inputs_Channel_385E794A;
	{attribute addProperty Name "EPM_Inputs_Channel_4"}
	EPM_Inputs_Channel_4 : EPM_Inputs_Channel_385E794A;
	{attribute addProperty Name "EPM_Inputs_Channel_5"}
	EPM_Inputs_Channel_5 : EPM_Inputs_Channel_385E794A;
	{attribute addProperty Name "EPM_Inputs_Channel_6"}
	EPM_Inputs_Channel_6 : EPM_Inputs_Channel_385E794A;
	{attribute addProperty Name "EPM_Inputs_Channel_7"}
	EPM_Inputs_Channel_7 : EPM_Inputs_Channel_385E794A;
	{attribute addProperty Name "EPM_Inputs_Channel_8"}
	EPM_Inputs_Channel_8 : EPM_Inputs_Channel_385E794A;
	{attribute addProperty Name "EPM_Inputs_Channel_9"}
	EPM_Inputs_Channel_9 : EPM_Inputs_Channel_385E794A;
	{attribute addProperty Name "EPM_Inputs_Channel_10"}
	EPM_Inputs_Channel_10 : EPM_Inputs_Channel_385E794A;
	{attribute addProperty Name "WcState"}
	WcState : WcState_9091E0EB;
	{attribute addProperty Name "InfoData"}
	InfoData : InfoData_32EB74EA;
END_STRUCT
END_TYPE

// ---- DUTs/IO/Boxes/CX1100_1FC0878B.TcDUT
{attribute 'GeneratedUsingTerminal: CX1100-0004-0000'}
{attribute addProperty BoxType "CX1100-0004-0000"}
{attribute addProperty Description "CX1100-0004 EtherCAT Power supply (2A E-Bus)"}
{attribute addProperty Physics "YKY"}
{attribute addProperty Id "InfoDataAT %I*InfoData_6F19DB2B2"}
{attribute addProperty CRC "532711307"}
{attribute addProperty Size "2"}
TYPE CX1100_1FC0878B EXTENDS EtcSlaveBoxBase_77A0E4A7 :
STRUCT
	{attribute addProperty Name "InfoData"}
	InfoData : InfoData_6F19DB2B;
END_STRUCT
END_TYPE

// ---- DUTs/IO/Boxes/CX5010_EtherCAT_slave_FEF7A27A.TcDUT
{attribute 'GeneratedUsingTerminal: CX5010 EtherCAT slave-1b82-0016'}
{attribute addProperty BoxType "CX5010 EtherCAT slave-1b82-0016"}
{attribute addProperty Description "CX5010 EtherCAT slave"}
{attribute addProperty Physics "YY"}
{attribute addProperty Id "IO_InputsEMPTY_STRUCTURE0Device_Status_MappingAT %I*Device_Status_Mapping_61F790772IO_OutputsEMPTY_STRUCTURE0WcStateAT %I*WcState_9091E0EB2InfoDataAT %I*InfoData_90184F0C16"}
{attribute addProperty CRC "4277641850"}
{attribute addProperty Size "20"}
TYPE CX5010_EtherCAT_slave_FEF7A27A EXTENDS EtcSlaveBoxBase_77A0E4A7 :
STRUCT
	{attribute addProperty Name "IO_Inputs"}
	IO_Inputs : EMPTY_STRUCTURE;
	{attribute addProperty Name "Device_Status_Mapping"}
	Device_Status_Mapping : Device_Status_Mapping_61F79077;
	{attribute addProperty Name "IO_Outputs"}
	IO_Outputs : EMPTY_STRUCTURE;
	{attribute addProperty Name "WcState"}
	WcState : WcState_9091E0EB;
	{attribute addProperty Name "InfoData"}
	InfoData : InfoData_90184F0C;
END_STRUCT
END_TYPE

// ---- DUTs/IO/Boxes/CX5020_EtherCAT_slave_FEF7A27A.TcDUT
{attribute 'GeneratedUsingTerminal: CX5020 EtherCAT slave-1b82-0016'}
{attribute addProperty BoxType "CX5020 EtherCAT slave-1b82-0016"}
{attribute addProperty Description "CX5020 EtherCAT slave"}
{attribute addProperty Physics "YY"}
{attribute addProperty Id "IO_InputsEMPTY_STRUCTURE0Device_Status_MappingAT %I*Device_Status_Mapping_61F790772IO_OutputsEMPTY_STRUCTURE0WcStateAT %I*WcState_9091E0EB2InfoDataAT %I*InfoData_90184F0C16"}
{attribute addProperty CRC "4277641850"}
{attribute addProperty Size "20"}
TYPE CX5020_EtherCAT_slave_FEF7A27A EXTENDS EtcSlaveBoxBase_77A0E4A7 :
STRUCT
	{attribute addProperty Name "IO_Inputs"}
	IO_Inputs : EMPTY_STRUCTURE;
	{attribute addProperty Name "Device_Status_Mapping"}
	Device_Status_Mapping : Device_Status_Mapping_61F79077;
	{attribute addProperty Name "IO_Outputs"}
	IO_Outputs : EMPTY_STRUCTURE;
	{attribute addProperty Name "WcState"}
	WcState : WcState_9091E0EB;
	{attribute addProperty Name "InfoData"}
	InfoData : InfoData_90184F0C;
END_STRUCT
END_TYPE

// ---- DUTs/IO/Boxes/CX8010_EtherCAT_slave_FEF7A27A.TcDUT
{attribute 'GeneratedUsingTerminal: CX8010 EtherCAT slave-0000-0016'}
{attribute addProperty BoxType "CX8010 EtherCAT slave-0000-0016"}
{attribute addProperty Description "CX8010 EtherCAT slave"}
{attribute addProperty Physics "YY"}
{attribute addProperty Id "IO_InputsEMPTY_STRUCTURE0Device_Status_MappingAT %I*Device_Status_Mapping_61F790772IO_OutputsEMPTY_STRUCTURE0WcStateAT %I*WcState_9091E0EB2InfoDataAT %I*InfoData_90184F0C16"}
{attribute addProperty CRC "4277641850"}
{attribute addProperty Size "20"}
TYPE CX8010_EtherCAT_slave_FEF7A27A EXTENDS EtcSlaveBoxBase_77A0E4A7 :
STRUCT
	{attribute addProperty Name "IO_Inputs"}
	IO_Inputs : EMPTY_STRUCTURE;
	{attribute addProperty Name "Device_Status_Mapping"}
	Device_Status_Mapping : Device_Status_Mapping_61F79077;
	{attribute addProperty Name "IO_Outputs"}
	IO_Outputs : EMPTY_STRUCTURE;
	{attribute addProperty Name "WcState"}
	WcState : WcState_9091E0EB;
	{attribute addProperty Name "InfoData"}
	InfoData : InfoData_90184F0C;
END_STRUCT
END_TYPE

// ---- DUTs/IO/Boxes/CX8110_EtherCAT_slave_FEF7A27A.TcDUT
{attribute 'GeneratedUsingTerminal: CX8110 EtherCAT slave-0000-0016'}
{attribute addProperty BoxType "CX8110 EtherCAT slave-0000-0016"}
{attribute addProperty Description "CX8110 EtherCAT slave"}
{attribute addProperty Physics "YY"}
{attribute addProperty Id "IO_InputsEMPTY_STRUCTURE0Device_Status_MappingAT %I*Device_Status_Mapping_61F790772IO_OutputsEMPTY_STRUCTURE0WcStateAT %I*WcState_9091E0EB2InfoDataAT %I*InfoData_90184F0C16"}
{attribute addProperty CRC "4277641850"}
{attribute addProperty Size "20"}
TYPE CX8110_EtherCAT_slave_FEF7A27A EXTENDS EtcSlaveBoxBase_77A0E4A7 :
STRUCT
	{attribute addProperty Name "IO_Inputs"}
	IO_Inputs : EMPTY_STRUCTURE;
	{attribute addProperty Name "Device_Status_Mapping"}
	Device_Status_Mapping : Device_Status_Mapping_61F79077;
	{attribute addProperty Name "IO_Outputs"}
	IO_Outputs : EMPTY_STRUCTURE;
	{attribute addProperty Name "WcState"}
	WcState : WcState_9091E0EB;
	{attribute addProperty Name "InfoData"}
	InfoData : InfoData_90184F0C;
END_STRUCT
END_TYPE

// ---- DUTs/IO/Boxes/CX2020_EtherCAT_slave_FEF7A27A.TcDUT
{attribute 'GeneratedUsingTerminal: CX2020 EtherCAT slave-1b82-0016'}
{attribute addProperty BoxType "CX2020 EtherCAT slave-1b82-0016"}
{attribute addProperty Description "CX2020 EtherCAT slave"}
{attribute addProperty Physics "YY"}
{attribute addProperty Id "IO_InputsEMPTY_STRUCTURE0Device_Status_MappingAT %I*Device_Status_Mapping_61F790772IO_OutputsEMPTY_STRUCTURE0WcStateAT %I*WcState_9091E0EB2InfoDataAT %I*InfoData_90184F0C16"}
{attribute addProperty CRC "4277641850"}
{attribute addProperty Size "20"}
TYPE CX2020_EtherCAT_slave_FEF7A27A EXTENDS EtcSlaveBoxBase_77A0E4A7 :
STRUCT
	{attribute addProperty Name "IO_Inputs"}
	IO_Inputs : EMPTY_STRUCTURE;
	{attribute addProperty Name "Device_Status_Mapping"}
	Device_Status_Mapping : Device_Status_Mapping_61F79077;
	{attribute addProperty Name "IO_Outputs"}
	IO_Outputs : EMPTY_STRUCTURE;
	{attribute addProperty Name "WcState"}
	WcState : WcState_9091E0EB;
	{attribute addProperty Name "InfoData"}
	InfoData : InfoData_90184F0C;
END_STRUCT
END_TYPE

// ---- DUTs/IO/Boxes/CX2030_EtherCAT_slave_FEF7A27A.TcDUT
{attribute 'GeneratedUsingTerminal: CX2030 EtherCAT slave-1b82-0016'}
{attribute addProperty BoxType "CX2030 EtherCAT slave-1b82-0016"}
{attribute addProperty Description "CX2030 EtherCAT slave"}
{attribute addProperty Physics "YY"}
{attribute addProperty Id "IO_InputsEMPTY_STRUCTURE0Device_Status_MappingAT %I*Device_Status_Mapping_61F790772IO_OutputsEMPTY_STRUCTURE0WcStateAT %I*WcState_9091E0EB2InfoDataAT %I*InfoData_90184F0C16"}
{attribute addProperty CRC "4277641850"}
{attribute addProperty Size "20"}
TYPE CX2030_EtherCAT_slave_FEF7A27A EXTENDS EtcSlaveBoxBase_77A0E4A7 :
STRUCT
	{attribute addProperty Name "IO_Inputs"}
	IO_Inputs : EMPTY_STRUCTURE;
	{attribute addProperty Name "Device_Status_Mapping"}
	Device_Status_Mapping : Device_Status_Mapping_61F79077;
	{attribute addProperty Name "IO_Outputs"}
	IO_Outputs : EMPTY_STRUCTURE;
	{attribute addProperty Name "WcState"}
	WcState : WcState_9091E0EB;
	{attribute addProperty Name "InfoData"}
	InfoData : InfoData_90184F0C;
END_STRUCT
END_TYPE

// ---- DUTs/IO/Boxes/CX2033_EtherCAT_slave_FEF7A27A.TcDUT
{attribute 'GeneratedUsingTerminal: CX2033 EtherCAT slave-1b82-0016'}
{attribute addProperty BoxType "CX2033 EtherCAT slave-1b82-0016"}
{attribute addProperty Description "CX2033 EtherCAT slave"}
{attribute addProperty Physics "YY"}
{attribute addProperty Id "IO_InputsEMPTY_STRUCTURE0Device_Status_MappingAT %I*Device_Status_Mapping_61F790772IO_OutputsEMPTY_STRUCTURE0WcStateAT %I*WcState_9091E0EB2InfoDataAT %I*InfoData_90184F0C16"}
{attribute addProperty CRC "4277641850"}
{attribute addProperty Size "20"}
TYPE CX2033_EtherCAT_slave_FEF7A27A EXTENDS EtcSlaveBoxBase_77A0E4A7 :
STRUCT
	{attribute addProperty Name "IO_Inputs"}
	IO_Inputs : EMPTY_STRUCTURE;
	{attribute addProperty Name "Device_Status_Mapping"}
	Device_Status_Mapping : Device_Status_Mapping_61F79077;
	{attribute addProperty Name "IO_Outputs"}
	IO_Outputs : EMPTY_STRUCTURE;
	{attribute addProperty Name "WcState"}
	WcState : WcState_9091E0EB;
	{attribute addProperty Name "InfoData"}
	InfoData : InfoData_90184F0C;
END_STRUCT
END_TYPE

// ---- DUTs/IO/Boxes/CX2040_EtherCAT_slave_FEF7A27A.TcDUT
{attribute 'GeneratedUsingTerminal: CX2040 EtherCAT slave-1b82-0016'}
{attribute addProperty BoxType "CX2040 EtherCAT slave-1b82-0016"}
{attribute addProperty Description "CX2040 EtherCAT slave"}
{attribute addProperty Physics "YY"}
{attribute addProperty Id "IO_InputsEMPTY_STRUCTURE0Device_Status_MappingAT %I*Device_Status_Mapping_61F790772IO_OutputsEMPTY_STRUCTURE0WcStateAT %I*WcState_9091E0EB2InfoDataAT %I*InfoData_90184F0C16"}
{attribute addProperty CRC "4277641850"}
{attribute addProperty Size "20"}
TYPE CX2040_EtherCAT_slave_FEF7A27A EXTENDS EtcSlaveBoxBase_77A0E4A7 :
STRUCT
	{attribute addProperty Name "IO_Inputs"}
	IO_Inputs : EMPTY_STRUCTURE;
	{attribute addProperty Name "Device_Status_Mapping"}
	Device_Status_Mapping : Device_Status_Mapping_61F79077;
	{attribute addProperty Name "IO_Outputs"}
	IO_Outputs : EMPTY_STRUCTURE;
	{attribute addProperty Name "WcState"}
	WcState : WcState_9091E0EB;
	{attribute addProperty Name "InfoData"}
	InfoData : InfoData_90184F0C;
END_STRUCT
END_TYPE

// ---- DUTs/IO/Boxes/CX2042_EtherCAT_slave_FEF7A27A.TcDUT
{attribute 'GeneratedUsingTerminal: CX2042 EtherCAT slave-1b82-0016'}
{attribute addProperty BoxType "CX2042 EtherCAT slave-1b82-0016"}
{attribute addProperty Description "CX2042 EtherCAT slave"}
{attribute addProperty Physics "YY"}
{attribute addProperty Id "IO_InputsEMPTY_STRUCTURE0Device_Status_MappingAT %I*Device_Status_Mapping_61F790772IO_OutputsEMPTY_STRUCTURE0WcStateAT %I*WcState_9091E0EB2InfoDataAT %I*InfoData_90184F0C16"}
{attribute addProperty CRC "4277641850"}
{attribute addProperty Size "20"}
TYPE CX2042_EtherCAT_slave_FEF7A27A EXTENDS EtcSlaveBoxBase_77A0E4A7 :
STRUCT
	{attribute addProperty Name "IO_Inputs"}
	IO_Inputs : EMPTY_STRUCTURE;
	{attribute addProperty Name "Device_Status_Mapping"}
	Device_Status_Mapping : Device_Status_Mapping_61F79077;
	{attribute addProperty Name "IO_Outputs"}
	IO_Outputs : EMPTY_STRUCTURE;
	{attribute addProperty Name "WcState"}
	WcState : WcState_9091E0EB;
	{attribute addProperty Name "InfoData"}
	InfoData : InfoData_90184F0C;
END_STRUCT
END_TYPE

// ---- DUTs/IO/Boxes/CX2043_EtherCAT_slave_FEF7A27A.TcDUT
{attribute 'GeneratedUsingTerminal: CX2043 EtherCAT slave-1b82-0016'}
{attribute addProperty BoxType "CX2043 EtherCAT slave-1b82-0016"}
{attribute addProperty Description "CX2043 EtherCAT slave"}
{attribute addProperty Physics "YY"}
{attribute addProperty Id "IO_InputsEMPTY_STRUCTURE0Device_Status_MappingAT %I*Device_Status_Mapping_61F790772IO_OutputsEMPTY_STRUCTURE0WcStateAT %I*WcState_9091E0EB2InfoDataAT %I*InfoData_90184F0C16"}
{attribute addProperty CRC "4277641850"}
{attribute addProperty Size "20"}
TYPE CX2043_EtherCAT_slave_FEF7A27A EXTENDS EtcSlaveBoxBase_77A0E4A7 :
STRUCT
	{attribute addProperty Name "IO_Inputs"}
	IO_Inputs : EMPTY_STRUCTURE;
	{attribute addProperty Name "Device_Status_Mapping"}
	Device_Status_Mapping : Device_Status_Mapping_61F79077;
	{attribute addProperty Name "IO_Outputs"}
	IO_Outputs : EMPTY_STRUCTURE;
	{attribute addProperty Name "WcState"}
	WcState : WcState_9091E0EB;
	{attribute addProperty Name "InfoData"}
	InfoData : InfoData_90184F0C;
END_STRUCT
END_TYPE

// ---- DUTs/IO/Boxes/CX2062_EtherCAT_slave_FEF7A27A.TcDUT
{attribute 'GeneratedUsingTerminal: CX2062 EtherCAT slave-1b82-0016'}
{attribute addProperty BoxType "CX2062 EtherCAT slave-1b82-0016"}
{attribute addProperty Description "CX2062 EtherCAT slave"}
{attribute addProperty Physics "YY"}
{attribute addProperty Id "IO_InputsEMPTY_STRUCTURE0Device_Status_MappingAT %I*Device_Status_Mapping_61F790772IO_OutputsEMPTY_STRUCTURE0WcStateAT %I*WcState_9091E0EB2InfoDataAT %I*InfoData_90184F0C16"}
{attribute addProperty CRC "4277641850"}
{attribute addProperty Size "20"}
TYPE CX2062_EtherCAT_slave_FEF7A27A EXTENDS EtcSlaveBoxBase_77A0E4A7 :
STRUCT
	{attribute addProperty Name "IO_Inputs"}
	IO_Inputs : EMPTY_STRUCTURE;
	{attribute addProperty Name "Device_Status_Mapping"}
	Device_Status_Mapping : Device_Status_Mapping_61F79077;
	{attribute addProperty Name "IO_Outputs"}
	IO_Outputs : EMPTY_STRUCTURE;
	{attribute addProperty Name "WcState"}
	WcState : WcState_9091E0EB;
	{attribute addProperty Name "InfoData"}
	InfoData : InfoData_90184F0C;
END_STRUCT
END_TYPE

// ---- DUTs/IO/Boxes/CX2072_EtherCAT_slave_FEF7A27A.TcDUT
{attribute 'GeneratedUsingTerminal: CX2072 EtherCAT slave-1b82-0016'}
{attribute addProperty BoxType "CX2072 EtherCAT slave-1b82-0016"}
{attribute addProperty Description "CX2072 EtherCAT slave"}
{attribute addProperty Physics "YY"}
{attribute addProperty Id "IO_InputsEMPTY_STRUCTURE0Device_Status_MappingAT %I*Device_Status_Mapping_61F790772IO_OutputsEMPTY_STRUCTURE0WcStateAT %I*WcState_9091E0EB2InfoDataAT %I*InfoData_90184F0C16"}
{attribute addProperty CRC "4277641850"}
{attribute addProperty Size "20"}
TYPE CX2072_EtherCAT_slave_FEF7A27A EXTENDS EtcSlaveBoxBase_77A0E4A7 :
STRUCT
	{attribute addProperty Name "IO_Inputs"}
	IO_Inputs : EMPTY_STRUCTURE;
	{attribute addProperty Name "Device_Status_Mapping"}
	Device_Status_Mapping : Device_Status_Mapping_61F79077;
	{attribute addProperty Name "IO_Outputs"}
	IO_Outputs : EMPTY_STRUCTURE;
	{attribute addProperty Name "WcState"}
	WcState : WcState_9091E0EB;
	{attribute addProperty Name "InfoData"}
	InfoData : InfoData_90184F0C;
END_STRUCT
END_TYPE

// ---- DUTs/IO/Boxes/CX9020_EtherCAT_slave_FEF7A27A.TcDUT
{attribute 'GeneratedUsingTerminal: CX9020 EtherCAT slave-1b82-0016'}
{attribute addProperty BoxType "CX9020 EtherCAT slave-1b82-0016"}
{attribute addProperty Description "CX9020 EtherCAT slave"}
{attribute addProperty Physics "YY"}
{attribute addProperty Id "IO_InputsEMPTY_STRUCTURE0Device_Status_MappingAT %I*Device_Status_Mapping_61F790772IO_OutputsEMPTY_STRUCTURE0WcStateAT %I*WcState_9091E0EB2InfoDataAT %I*InfoData_90184F0C16"}
{attribute addProperty CRC "4277641850"}
{attribute addProperty Size "20"}
TYPE CX9020_EtherCAT_slave_FEF7A27A EXTENDS EtcSlaveBoxBase_77A0E4A7 :
STRUCT
	{attribute addProperty Name "IO_Inputs"}
	IO_Inputs : EMPTY_STRUCTURE;
	{attribute addProperty Name "Device_Status_Mapping"}
	Device_Status_Mapping : Device_Status_Mapping_61F79077;
	{attribute addProperty Name "IO_Outputs"}
	IO_Outputs : EMPTY_STRUCTURE;
	{attribute addProperty Name "WcState"}
	WcState : WcState_9091E0EB;
	{attribute addProperty Name "InfoData"}
	InfoData : InfoData_90184F0C;
END_STRUCT
END_TYPE

// ---- DUTs/IO/Boxes/CX5120_EtherCAT_slave_FEF7A27A.TcDUT
{attribute 'GeneratedUsingTerminal: CX5120 EtherCAT slave-1b82-0016'}
{attribute addProperty BoxType "CX5120 EtherCAT slave-1b82-0016"}
{attribute addProperty Description "CX5120 EtherCAT slave"}
{attribute addProperty Physics "YY"}
{attribute addProperty Id "IO_InputsEMPTY_STRUCTURE0Device_Status_MappingAT %I*Device_Status_Mapping_61F790772IO_OutputsEMPTY_STRUCTURE0WcStateAT %I*WcState_9091E0EB2InfoDataAT %I*InfoData_90184F0C16"}
{attribute addProperty CRC "4277641850"}
{attribute addProperty Size "20"}
TYPE CX5120_EtherCAT_slave_FEF7A27A EXTENDS EtcSlaveBoxBase_77A0E4A7 :
STRUCT
	{attribute addProperty Name "IO_Inputs"}
	IO_Inputs : EMPTY_STRUCTURE;
	{attribute addProperty Name "Device_Status_Mapping"}
	Device_Status_Mapping : Device_Status_Mapping_61F79077;
	{attribute addProperty Name "IO_Outputs"}
	IO_Outputs : EMPTY_STRUCTURE;
	{attribute addProperty Name "WcState"}
	WcState : WcState_9091E0EB;
	{attribute addProperty Name "InfoData"}
	InfoData : InfoData_90184F0C;
END_STRUCT
END_TYPE

// ---- DUTs/IO/Boxes/CX5130_EtherCAT_slave_FEF7A27A.TcDUT
{attribute 'GeneratedUsingTerminal: CX5130 EtherCAT slave-1b82-0016'}
{attribute addProperty BoxType "CX5130 EtherCAT slave-1b82-0016"}
{attribute addProperty Description "CX5130 EtherCAT slave"}
{attribute addProperty Physics "YY"}
{attribute addProperty Id "IO_InputsEMPTY_STRUCTURE0Device_Status_MappingAT %I*Device_Status_Mapping_61F790772IO_OutputsEMPTY_STRUCTURE0WcStateAT %I*WcState_9091E0EB2InfoDataAT %I*InfoData_90184F0C16"}
{attribute addProperty CRC "4277641850"}
{attribute addProperty Size "20"}
TYPE CX5130_EtherCAT_slave_FEF7A27A EXTENDS EtcSlaveBoxBase_77A0E4A7 :
STRUCT
	{attribute addProperty Name "IO_Inputs"}
	IO_Inputs : EMPTY_STRUCTURE;
	{attribute addProperty Name "Device_Status_Mapping"}
	Device_Status_Mapping : Device_Status_Mapping_61F79077;
	{attribute addProperty Name "IO_Outputs"}
	IO_Outputs : EMPTY_STRUCTURE;
	{attribute addProperty Name "WcState"}
	WcState : WcState_9091E0EB;
	{attribute addProperty Name "InfoData"}
	InfoData : InfoData_90184F0C;
END_STRUCT
END_TYPE

// ---- DUTs/IO/Boxes/CX5140_EtherCAT_slave_FEF7A27A.TcDUT
{attribute 'GeneratedUsingTerminal: CX5140 EtherCAT slave-1b82-0016'}
{attribute addProperty BoxType "CX5140 EtherCAT slave-1b82-0016"}
{attribute addProperty Description "CX5140 EtherCAT slave"}
{attribute addProperty Physics "YY"}
{attribute addProperty Id "IO_InputsEMPTY_STRUCTURE0Device_Status_MappingAT %I*Device_Status_Mapping_61F790772IO_OutputsEMPTY_STRUCTURE0WcStateAT %I*WcState_9091E0EB2InfoDataAT %I*InfoData_90184F0C16"}
{attribute addProperty CRC "4277641850"}
{attribute addProperty Size "20"}
TYPE CX5140_EtherCAT_slave_FEF7A27A EXTENDS EtcSlaveBoxBase_77A0E4A7 :
STRUCT
	{attribute addProperty Name "IO_Inputs"}
	IO_Inputs : EMPTY_STRUCTURE;
	{attribute addProperty Name "Device_Status_Mapping"}
	Device_Status_Mapping : Device_Status_Mapping_61F79077;
	{attribute addProperty Name "IO_Outputs"}
	IO_Outputs : EMPTY_STRUCTURE;
	{attribute addProperty Name "WcState"}
	WcState : WcState_9091E0EB;
	{attribute addProperty Name "InfoData"}
	InfoData : InfoData_90184F0C;
END_STRUCT
END_TYPE

// ---- DUTs/IO/Boxes/CX5230_EtherCAT_slave_FEF7A27A.TcDUT
{attribute 'GeneratedUsingTerminal: CX5230 EtherCAT slave-1b82-0016'}
{attribute addProperty BoxType "CX5230 EtherCAT slave-1b82-0016"}
{attribute addProperty Description "CX5230 EtherCAT slave"}
{attribute addProperty Physics "YY"}
{attribute addProperty Id "IO_InputsEMPTY_STRUCTURE0Device_Status_MappingAT %I*Device_Status_Mapping_61F790772IO_OutputsEMPTY_STRUCTURE0WcStateAT %I*WcState_9091E0EB2InfoDataAT %I*InfoData_90184F0C16"}
{attribute addProperty CRC "4277641850"}
{attribute addProperty Size "20"}
TYPE CX5230_EtherCAT_slave_FEF7A27A EXTENDS EtcSlaveBoxBase_77A0E4A7 :
STRUCT
	{attribute addProperty Name "IO_Inputs"}
	IO_Inputs : EMPTY_STRUCTURE;
	{attribute addProperty Name "Device_Status_Mapping"}
	Device_Status_Mapping : Device_Status_Mapping_61F79077;
	{attribute addProperty Name "IO_Outputs"}
	IO_Outputs : EMPTY_STRUCTURE;
	{attribute addProperty Name "WcState"}
	WcState : WcState_9091E0EB;
	{attribute addProperty Name "InfoData"}
	InfoData : InfoData_90184F0C;
END_STRUCT
END_TYPE

// ---- DUTs/IO/Boxes/CX5240_EtherCAT_slave_FEF7A27A.TcDUT
{attribute 'GeneratedUsingTerminal: CX5240 EtherCAT slave-1b82-0016'}
{attribute addProperty BoxType "CX5240 EtherCAT slave-1b82-0016"}
{attribute addProperty Description "CX5240 EtherCAT slave"}
{attribute addProperty Physics "YY"}
{attribute addProperty Id "IO_InputsEMPTY_STRUCTURE0Device_Status_MappingAT %I*Device_Status_Mapping_61F790772IO_OutputsEMPTY_STRUCTURE0WcStateAT %I*WcState_9091E0EB2InfoDataAT %I*InfoData_90184F0C16"}
{attribute addProperty CRC "4277641850"}
{attribute addProperty Size "20"}
TYPE CX5240_EtherCAT_slave_FEF7A27A EXTENDS EtcSlaveBoxBase_77A0E4A7 :
STRUCT
	{attribute addProperty Name "IO_Inputs"}
	IO_Inputs : EMPTY_STRUCTURE;
	{attribute addProperty Name "Device_Status_Mapping"}
	Device_Status_Mapping : Device_Status_Mapping_61F79077;
	{attribute addProperty Name "IO_Outputs"}
	IO_Outputs : EMPTY_STRUCTURE;
	{attribute addProperty Name "WcState"}
	WcState : WcState_9091E0EB;
	{attribute addProperty Name "InfoData"}
	InfoData : InfoData_90184F0C;
END_STRUCT
END_TYPE

// ---- DUTs/IO/Boxes/KL_5E2F016F.TcDUT
{attribute 'GeneratedUsingTerminal: KL9976-0050'}
{attribute addProperty BoxType "KL9976-0050"}
{attribute addProperty Description ""}
{attribute addProperty Physics ""}
{attribute addProperty Id "Channel_1AT %I*0"}
{attribute addProperty CRC "1580138863"}
{attribute addProperty Size "0"}
TYPE KL_5E2F016F :
STRUCT
	{attribute addProperty Name "Channel_1"}
	Channel_1 : ;
END_STRUCT
END_TYPE

// ---- DUTs/IO/Boxes/KL_2EA97E3E.TcDUT
{attribute 'GeneratedUsingTerminal: KL9940-0050'}
{attribute addProperty BoxType "KL9940-0050"}
{attribute addProperty Description ""}
{attribute addProperty Physics ""}
{attribute addProperty Id "Channel_1AT %I*Channel_954C2EED0"}
{attribute addProperty CRC "782859838"}
{attribute addProperty Size "0"}
TYPE KL_2EA97E3E :
STRUCT
	{attribute addProperty Name "Channel_1"}
	Channel_1 : Channel_954C2EED;
END_STRUCT
END_TYPE

// ---- DUTs/IO/Boxes/KL_1187B721.TcDUT
{attribute 'GeneratedUsingTerminal: KL9900-0054'}
{attribute addProperty BoxType "KL9900-0054"}
{attribute addProperty Description ""}
{attribute addProperty Physics ""}
{attribute addProperty Id "Channel_1AT %Q*Channel_60E28ED20"}
{attribute addProperty CRC "294106913"}
{attribute addProperty Size "0"}
TYPE KL_1187B721 :
STRUCT
	{attribute addProperty Name "Channel_1"}
	Channel_1 : Channel_60E28ED2;
END_STRUCT
END_TYPE

// ---- DUTs/IO/Boxes/KL_E991A364.TcDUT
{attribute 'GeneratedUsingTerminal: KL9900-0055'}
{attribute addProperty BoxType "KL9900-0055"}
{attribute addProperty Description ""}
{attribute addProperty Physics ""}
{attribute addProperty Id "Channel_1AT %Q*Channel_7DE261950"}
{attribute addProperty CRC "3918635876"}
{attribute addProperty Size "0"}
TYPE KL_E991A364 :
STRUCT
	{attribute addProperty Name "Channel_1"}
	Channel_1 : Channel_7DE26195;
END_STRUCT
END_TYPE

// ---- DUTs/IO/Boxes/KL_063F0990.TcDUT
{attribute 'GeneratedUsingTerminal: KL9900-0056'}
{attribute addProperty BoxType "KL9900-0056"}
{attribute addProperty Description ""}
{attribute addProperty Physics ""}
{attribute addProperty Id "Channel_1AT %Q*Channel_2E0D480D0"}
{attribute addProperty CRC "104794512"}
{attribute addProperty Size "0"}
TYPE KL_063F0990 :
STRUCT
	{attribute addProperty Name "Channel_1"}
	Channel_1 : Channel_2E0D480D;
END_STRUCT
END_TYPE

// ---- DUTs/IO/Boxes/KL_5AE00A1C.TcDUT
{attribute 'GeneratedUsingTerminal: KL9900-0057'}
{attribute addProperty BoxType "KL9900-0057"}
{attribute addProperty Description ""}
{attribute addProperty Physics ""}
{attribute addProperty Id "Channel_1AT %Q*Channel_61FC15360"}
{attribute addProperty CRC "1524632092"}
{attribute addProperty Size "0"}
TYPE KL_5AE00A1C :
STRUCT
	{attribute addProperty Name "Channel_1"}
	Channel_1 : Channel_61FC1536;
END_STRUCT
END_TYPE

// ---- DUTs/IO/Boxes/KL_CFA8830D.TcDUT
{attribute 'GeneratedUsingTerminal: KL9900-0058'}
{attribute addProperty BoxType "KL9900-0058"}
{attribute addProperty Description ""}
{attribute addProperty Physics ""}
{attribute addProperty Id "Channel_1AT %Q*Channel_16463F740"}
{attribute addProperty CRC "3483927309"}
{attribute addProperty Size "0"}
TYPE KL_CFA8830D :
STRUCT
	{attribute addProperty Name "Channel_1"}
	Channel_1 : Channel_16463F74;
END_STRUCT
END_TYPE

// ---- DUTs/IO/Boxes/KL_DBC0B844.TcDUT
{attribute 'GeneratedUsingTerminal: KL9900-0059'}
{attribute addProperty BoxType "KL9900-0059"}
{attribute addProperty Description ""}
{attribute addProperty Physics ""}
{attribute addProperty Id "Channel_1AT %Q*Channel_707BD1FE0"}
{attribute addProperty CRC "3686840388"}
{attribute addProperty Size "0"}
TYPE KL_DBC0B844 :
STRUCT
	{attribute addProperty Name "Channel_1"}
	Channel_1 : Channel_707BD1FE;
END_STRUCT
END_TYPE

// ---- DUTs/IO/Boxes/KL_6930B3B2.TcDUT
{attribute 'GeneratedUsingTerminal: KL9900-0060'}
{attribute addProperty BoxType "KL9900-0060"}
{attribute addProperty Description ""}
{attribute addProperty Physics ""}
{attribute addProperty Id "Channel_1AT %Q*Channel_7D202F580"}
{attribute addProperty CRC "1764799410"}
{attribute addProperty Size "0"}
TYPE KL_6930B3B2 :
STRUCT
	{attribute addProperty Name "Channel_1"}
	Channel_1 : Channel_7D202F58;
END_STRUCT
END_TYPE

// ---- DUTs/IO/Boxes/KL_4F0DAD84.TcDUT
{attribute 'GeneratedUsingTerminal: KL9900-0063'}
{attribute addProperty BoxType "KL9900-0063"}
{attribute addProperty Description ""}
{attribute addProperty Physics ""}
{attribute addProperty Id "Channel_1AT %Q*Channel_6CC0E2260"}
{attribute addProperty CRC "1326296452"}
{attribute addProperty Size "0"}
TYPE KL_4F0DAD84 :
STRUCT
	{attribute addProperty Name "Channel_1"}
	Channel_1 : Channel_6CC0E226;
END_STRUCT
END_TYPE

// ---- DUTs/IO/Boxes/KL_2227C35B.TcDUT
{attribute 'GeneratedUsingTerminal: KL9900-0064'}
{attribute addProperty BoxType "KL9900-0064"}
{attribute addProperty Description ""}
{attribute addProperty Physics ""}
{attribute addProperty Id "Channel_1AT %Q*Channel_0F0CD9400"}
{attribute addProperty CRC "573031259"}
{attribute addProperty Size "0"}
TYPE KL_2227C35B :
STRUCT
	{attribute addProperty Name "Channel_1"}
	Channel_1 : Channel_0F0CD940;
END_STRUCT
END_TYPE

// ---- DUTs/IO/Boxes/KL_E653A8C1.TcDUT
{attribute 'GeneratedUsingTerminal: KL9900-0062'}
{attribute addProperty BoxType "KL9900-0062"}
{attribute addProperty Description ""}
{attribute addProperty Physics ""}
{attribute addProperty Id "Channel_1AT %I*Channel_65B766000"}
{attribute addProperty CRC "3864242369"}
{attribute addProperty Size "0"}
TYPE KL_E653A8C1 :
STRUCT
	{attribute addProperty Name "Channel_1"}
	Channel_1 : Channel_65B76600;
END_STRUCT
END_TYPE

// ---- DUTs/IO/Boxes/KL1012_BB38DA8F.TcDUT
{attribute 'GeneratedUsingTerminal: KL1012'}
{attribute addProperty BoxType "KL1012"}
{attribute addProperty Description ""}
{attribute addProperty Physics ""}
{attribute addProperty Id "Channel_1AT %I*Channel_87C95E760Channel_2AT %I*Channel_87C95E760"}
{attribute addProperty CRC "3141065359"}
{attribute addProperty Size "0"}
TYPE KL1012_BB38DA8F :
STRUCT
	{attribute addProperty Name "Channel_1"}
	Channel_1 : Channel_87C95E76;
	{attribute addProperty Name "Channel_2"}
	Channel_2 : Channel_87C95E76;
END_STRUCT
END_TYPE

// ---- DUTs/IO/Boxes/KL1032_BB38DA8F.TcDUT
{attribute 'GeneratedUsingTerminal: KL1032'}
{attribute addProperty BoxType "KL1032"}
{attribute addProperty Description ""}
{attribute addProperty Physics ""}
{attribute addProperty Id "Channel_1AT %I*Channel_87C95E760Channel_2AT %I*Channel_87C95E760"}
{attribute addProperty CRC "3141065359"}
{attribute addProperty Size "0"}
TYPE KL1032_BB38DA8F :
STRUCT
	{attribute addProperty Name "Channel_1"}
	Channel_1 : Channel_87C95E76;
	{attribute addProperty Name "Channel_2"}
	Channel_2 : Channel_87C95E76;
END_STRUCT
END_TYPE

// ---- DUTs/IO/Boxes/KL1052_BB38DA8F.TcDUT
{attribute 'GeneratedUsingTerminal: KL1052'}
{attribute addProperty BoxType "KL1052"}
{attribute addProperty Description ""}
{attribute addProperty Physics ""}
{attribute addProperty Id "Channel_1AT %I*Channel_87C95E760Channel_2AT %I*Channel_87C95E760"}
{attribute addProperty CRC "3141065359"}
{attribute addProperty Size "0"}
TYPE KL1052_BB38DA8F :
STRUCT
	{attribute addProperty Name "Channel_1"}
	Channel_1 : Channel_87C95E76;
	{attribute addProperty Name "Channel_2"}
	Channel_2 : Channel_87C95E76;
END_STRUCT
END_TYPE

// ---- DUTs/IO/Boxes/KL1104_4A257D2B.TcDUT
{attribute 'GeneratedUsingTerminal: KL1104'}
{attribute addProperty BoxType "KL1104"}
{attribute addProperty Description ""}
{attribute addProperty Physics ""}
{attribute addProperty Id "Channel_1AT %I*Channel_87C95E760Channel_2AT %I*Channel_87C95E760Channel_3AT %I*Channel_87C95E760Channel_4AT %I*Channel_87C95E760"}
{attribute addProperty CRC "1243970859"}
{attribute addProperty Size "0"}
TYPE KL1104_4A257D2B :
STRUCT
	{attribute addProperty Name "Channel_1"}
	Channel_1 : Channel_87C95E76;
	{attribute addProperty Name "Channel_2"}
	Channel_2 : Channel_87C95E76;
	{attribute addProperty Name "Channel_3"}
	Channel_3 : Channel_87C95E76;
	{attribute addProperty Name "Channel_4"}
	Channel_4 : Channel_87C95E76;
END_STRUCT
END_TYPE

// ---- DUTs/IO/Boxes/KL1114_4A257D2B.TcDUT
{attribute 'GeneratedUsingTerminal: KL1114'}
{attribute addProperty BoxType "KL1114"}
{attribute addProperty Description ""}
{attribute addProperty Physics ""}
{attribute addProperty Id "Channel_1AT %I*Channel_87C95E760Channel_2AT %I*Channel_87C95E760Channel_3AT %I*Channel_87C95E760Channel_4AT %I*Channel_87C95E760"}
{attribute addProperty CRC "1243970859"}
{attribute addProperty Size "0"}
TYPE KL1114_4A257D2B :
STRUCT
	{attribute addProperty Name "Channel_1"}
	Channel_1 : Channel_87C95E76;
	{attribute addProperty Name "Channel_2"}
	Channel_2 : Channel_87C95E76;
	{attribute addProperty Name "Channel_3"}
	Channel_3 : Channel_87C95E76;
	{attribute addProperty Name "Channel_4"}
	Channel_4 : Channel_87C95E76;
END_STRUCT
END_TYPE

// ---- DUTs/IO/Boxes/KL1124_4A257D2B.TcDUT
{attribute 'GeneratedUsingTerminal: KL1124'}
{attribute addProperty BoxType "KL1124"}
{attribute addProperty Description ""}
{attribute addProperty Physics ""}
{attribute addProperty Id "Channel_1AT %I*Channel_87C95E760Channel_2AT %I*Channel_87C95E760Channel_3AT %I*Channel_87C95E760Channel_4AT %I*Channel_87C95E760"}
{attribute addProperty CRC "1243970859"}
{attribute addProperty Size "0"}
TYPE KL1124_4A257D2B :
STRUCT
	{attribute addProperty Name "Channel_1"}
	Channel_1 : Channel_87C95E76;
	{attribute addProperty Name "Channel_2"}
	Channel_2 : Channel_87C95E76;
	{attribute addProperty Name "Channel_3"}
	Channel_3 : Channel_87C95E76;
	{attribute addProperty Name "Channel_4"}
	Channel_4 : Channel_87C95E76;
END_STRUCT
END_TYPE

// ---- DUTs/IO/Boxes/KL1154_4A257D2B.TcDUT
{attribute 'GeneratedUsingTerminal: KL1154'}
{attribute addProperty BoxType "KL1154"}
{attribute addProperty Description ""}
{attribute addProperty Physics ""}
{attribute addProperty Id "Channel_1AT %I*Channel_87C95E760Channel_2AT %I*Channel_87C95E760Channel_3AT %I*Channel_87C95E760Channel_4AT %I*Channel_87C95E760"}
{attribute addProperty CRC "1243970859"}
{attribute addProperty Size "0"}
TYPE KL1154_4A257D2B :
STRUCT
	{attribute addProperty Name "Channel_1"}
	Channel_1 : Channel_87C95E76;
	{attribute addProperty Name "Channel_2"}
	Channel_2 : Channel_87C95E76;
	{attribute addProperty Name "Channel_3"}
	Channel_3 : Channel_87C95E76;
	{attribute addProperty Name "Channel_4"}
	Channel_4 : Channel_87C95E76;
END_STRUCT
END_TYPE

// ---- DUTs/IO/Boxes/KL1164_4A257D2B.TcDUT
{attribute 'GeneratedUsingTerminal: KL1164'}
{attribute addProperty BoxType "KL1164"}
{attribute addProperty Description ""}
{attribute addProperty Physics ""}
{attribute addProperty Id "Channel_1AT %I*Channel_87C95E760Channel_2AT %I*Channel_87C95E760Channel_3AT %I*Channel_87C95E760Channel_4AT %I*Channel_87C95E760"}
{attribute addProperty CRC "1243970859"}
{attribute addProperty Size "0"}
TYPE KL1164_4A257D2B :
STRUCT
	{attribute addProperty Name "Channel_1"}
	Channel_1 : Channel_87C95E76;
	{attribute addProperty Name "Channel_2"}
	Channel_2 : Channel_87C95E76;
	{attribute addProperty Name "Channel_3"}
	Channel_3 : Channel_87C95E76;
	{attribute addProperty Name "Channel_4"}
	Channel_4 : Channel_87C95E76;
END_STRUCT
END_TYPE

// ---- DUTs/IO/Boxes/KL1184_4A257D2B.TcDUT
{attribute 'GeneratedUsingTerminal: KL1184'}
{attribute addProperty BoxType "KL1184"}
{attribute addProperty Description ""}
{attribute addProperty Physics ""}
{attribute addProperty Id "Channel_1AT %I*Channel_87C95E760Channel_2AT %I*Channel_87C95E760Channel_3AT %I*Channel_87C95E760Channel_4AT %I*Channel_87C95E760"}
{attribute addProperty CRC "1243970859"}
{attribute addProperty Size "0"}
TYPE KL1184_4A257D2B :
STRUCT
	{attribute addProperty Name "Channel_1"}
	Channel_1 : Channel_87C95E76;
	{attribute addProperty Name "Channel_2"}
	Channel_2 : Channel_87C95E76;
	{attribute addProperty Name "Channel_3"}
	Channel_3 : Channel_87C95E76;
	{attribute addProperty Name "Channel_4"}
	Channel_4 : Channel_87C95E76;
END_STRUCT
END_TYPE

// ---- DUTs/IO/Boxes/KL1194_4A257D2B.TcDUT
{attribute 'GeneratedUsingTerminal: KL1194'}
{attribute addProperty BoxType "KL1194"}
{attribute addProperty Description ""}
{attribute addProperty Physics ""}
{attribute addProperty Id "Channel_1AT %I*Channel_87C95E760Channel_2AT %I*Channel_87C95E760Channel_3AT %I*Channel_87C95E760Channel_4AT %I*Channel_87C95E760"}
{attribute addProperty CRC "1243970859"}
{attribute addProperty Size "0"}
TYPE KL1194_4A257D2B :
STRUCT
	{attribute addProperty Name "Channel_1"}
	Channel_1 : Channel_87C95E76;
	{attribute addProperty Name "Channel_2"}
	Channel_2 : Channel_87C95E76;
	{attribute addProperty Name "Channel_3"}
	Channel_3 : Channel_87C95E76;
	{attribute addProperty Name "Channel_4"}
	Channel_4 : Channel_87C95E76;
END_STRUCT
END_TYPE

// ---- DUTs/IO/Boxes/KL1212_EC84F46C.TcDUT
{attribute 'GeneratedUsingTerminal: KL1212'}
{attribute addProperty BoxType "KL1212"}
{attribute addProperty Description ""}
{attribute addProperty Physics ""}
{attribute addProperty Id "Channel_1AT %Q*Channel_72DF63360Channel_2AT %Q*Channel_72DF63360"}
{attribute addProperty CRC "3968136300"}
{attribute addProperty Size "0"}
TYPE KL1212_EC84F46C :
STRUCT
	{attribute addProperty Name "Channel_1"}
	Channel_1 : Channel_72DF6336;
	{attribute addProperty Name "Channel_2"}
	Channel_2 : Channel_72DF6336;
END_STRUCT
END_TYPE

// ---- DUTs/IO/Boxes/KL1232_BB38DA8F.TcDUT
{attribute 'GeneratedUsingTerminal: KL1232'}
{attribute addProperty BoxType "KL1232"}
{attribute addProperty Description ""}
{attribute addProperty Physics ""}
{attribute addProperty Id "Channel_1AT %I*Channel_87C95E760Channel_2AT %I*Channel_87C95E760"}
{attribute addProperty CRC "3141065359"}
{attribute addProperty Size "0"}
TYPE KL1232_BB38DA8F :
STRUCT
	{attribute addProperty Name "Channel_1"}
	Channel_1 : Channel_87C95E76;
	{attribute addProperty Name "Channel_2"}
	Channel_2 : Channel_87C95E76;
END_STRUCT
END_TYPE

// ---- DUTs/IO/Boxes/KL1302_BB38DA8F.TcDUT
{attribute 'GeneratedUsingTerminal: KL1302'}
{attribute addProperty BoxType "KL1302"}
{attribute addProperty Description ""}
{attribute addProperty Physics ""}
{attribute addProperty Id "Channel_1AT %I*Channel_87C95E760Channel_2AT %I*Channel_87C95E760"}
{attribute addProperty CRC "3141065359"}
{attribute addProperty Size "0"}
TYPE KL1302_BB38DA8F :
STRUCT
	{attribute addProperty Name "Channel_1"}
	Channel_1 : Channel_87C95E76;
	{attribute addProperty Name "Channel_2"}
	Channel_2 : Channel_87C95E76;
END_STRUCT
END_TYPE

// ---- DUTs/IO/Boxes/KL1304_4A257D2B.TcDUT
{attribute 'GeneratedUsingTerminal: KL1304'}
{attribute addProperty BoxType "KL1304"}
{attribute addProperty Description ""}
{attribute addProperty Physics ""}
{attribute addProperty Id "Channel_1AT %I*Channel_87C95E760Channel_2AT %I*Channel_87C95E760Channel_3AT %I*Channel_87C95E760Channel_4AT %I*Channel_87C95E760"}
{attribute addProperty CRC "1243970859"}
{attribute addProperty Size "0"}
TYPE KL1304_4A257D2B :
STRUCT
	{attribute addProperty Name "Channel_1"}
	Channel_1 : Channel_87C95E76;
	{attribute addProperty Name "Channel_2"}
	Channel_2 : Channel_87C95E76;
	{attribute addProperty Name "Channel_3"}
	Channel_3 : Channel_87C95E76;
	{attribute addProperty Name "Channel_4"}
	Channel_4 : Channel_87C95E76;
END_STRUCT
END_TYPE

// ---- DUTs/IO/Boxes/KL1312_BB38DA8F.TcDUT
{attribute 'GeneratedUsingTerminal: KL1312'}
{attribute addProperty BoxType "KL1312"}
{attribute addProperty Description ""}
{attribute addProperty Physics ""}
{attribute addProperty Id "Channel_1AT %I*Channel_87C95E760Channel_2AT %I*Channel_87C95E760"}
{attribute addProperty CRC "3141065359"}
{attribute addProperty Size "0"}
TYPE KL1312_BB38DA8F :
STRUCT
	{attribute addProperty Name "Channel_1"}
	Channel_1 : Channel_87C95E76;
	{attribute addProperty Name "Channel_2"}
	Channel_2 : Channel_87C95E76;
END_STRUCT
END_TYPE

// ---- DUTs/IO/Boxes/KL1314_4A257D2B.TcDUT
{attribute 'GeneratedUsingTerminal: KL1314'}
{attribute addProperty BoxType "KL1314"}
{attribute addProperty Description ""}
{attribute addProperty Physics ""}
{attribute addProperty Id "Channel_1AT %I*Channel_87C95E760Channel_2AT %I*Channel_87C95E760Channel_3AT %I*Channel_87C95E760Channel_4AT %I*Channel_87C95E760"}
{attribute addProperty CRC "1243970859"}
{attribute addProperty Size "0"}
TYPE KL1314_4A257D2B :
STRUCT
	{attribute addProperty Name "Channel_1"}
	Channel_1 : Channel_87C95E76;
	{attribute addProperty Name "Channel_2"}
	Channel_2 : Channel_87C95E76;
	{attribute addProperty Name "Channel_3"}
	Channel_3 : Channel_87C95E76;
	{attribute addProperty Name "Channel_4"}
	Channel_4 : Channel_87C95E76;
END_STRUCT
END_TYPE

// ---- DUTs/IO/Boxes/KL1352_B54AC54D.TcDUT
{attribute 'GeneratedUsingTerminal: KL1352'}
{attribute addProperty BoxType "KL1352"}
{attribute addProperty Description ""}
{attribute addProperty Physics ""}
{attribute addProperty Id "Channel_1AT %I*Channel_22DCD6950Channel_2AT %I*Channel_22DCD6950"}
{attribute addProperty CRC "3041576269"}
{attribute addProperty Size "0"}
TYPE KL1352_B54AC54D :
STRUCT
	{attribute addProperty Name "Channel_1"}
	Channel_1 : Channel_22DCD695;
	{attribute addProperty Name "Channel_2"}
	Channel_2 : Channel_22DCD695;
END_STRUCT
END_TYPE

// ---- DUTs/IO/Boxes/KL1362_B54AC54D.TcDUT
{attribute 'GeneratedUsingTerminal: KL1362'}
{attribute addProperty BoxType "KL1362"}
{attribute addProperty Description ""}
{attribute addProperty Physics ""}
{attribute addProperty Id "Channel_1AT %I*Channel_22DCD6950Channel_2AT %I*Channel_22DCD6950"}
{attribute addProperty CRC "3041576269"}
{attribute addProperty Size "0"}
TYPE KL1362_B54AC54D :
STRUCT
	{attribute addProperty Name "Channel_1"}
	Channel_1 : Channel_22DCD695;
	{attribute addProperty Name "Channel_2"}
	Channel_2 : Channel_22DCD695;
END_STRUCT
END_TYPE

// ---- DUTs/IO/Boxes/KL1382_B54AC54D.TcDUT
{attribute 'GeneratedUsingTerminal: KL1382'}
{attribute addProperty BoxType "KL1382"}
{attribute addProperty Description ""}
{attribute addProperty Physics ""}
{attribute addProperty Id "Channel_1AT %I*Channel_22DCD6950Channel_2AT %I*Channel_22DCD6950"}
{attribute addProperty CRC "3041576269"}
{attribute addProperty Size "0"}
TYPE KL1382_B54AC54D :
STRUCT
	{attribute addProperty Name "Channel_1"}
	Channel_1 : Channel_22DCD695;
	{attribute addProperty Name "Channel_2"}
	Channel_2 : Channel_22DCD695;
END_STRUCT
END_TYPE

// ---- DUTs/IO/Boxes/KL1402_BB38DA8F.TcDUT
{attribute 'GeneratedUsingTerminal: KL1402'}
{attribute addProperty BoxType "KL1402"}
{attribute addProperty Description ""}
{attribute addProperty Physics ""}
{attribute addProperty Id "Channel_1AT %I*Channel_87C95E760Channel_2AT %I*Channel_87C95E760"}
{attribute addProperty CRC "3141065359"}
{attribute addProperty Size "0"}
TYPE KL1402_BB38DA8F :
STRUCT
	{attribute addProperty Name "Channel_1"}
	Channel_1 : Channel_87C95E76;
	{attribute addProperty Name "Channel_2"}
	Channel_2 : Channel_87C95E76;
END_STRUCT
END_TYPE

// ---- DUTs/IO/Boxes/KL1404_4A257D2B.TcDUT
{attribute 'GeneratedUsingTerminal: KL1404'}
{attribute addProperty BoxType "KL1404"}
{attribute addProperty Description ""}
{attribute addProperty Physics ""}
{attribute addProperty Id "Channel_1AT %I*Channel_87C95E760Channel_2AT %I*Channel_87C95E760Channel_3AT %I*Channel_87C95E760Channel_4AT %I*Channel_87C95E760"}
{attribute addProperty CRC "1243970859"}
{attribute addProperty Size "0"}
TYPE KL1404_4A257D2B :
STRUCT
	{attribute addProperty Name "Channel_1"}
	Channel_1 : Channel_87C95E76;
	{attribute addProperty Name "Channel_2"}
	Channel_2 : Channel_87C95E76;
	{attribute addProperty Name "Channel_3"}
	Channel_3 : Channel_87C95E76;
	{attribute addProperty Name "Channel_4"}
	Channel_4 : Channel_87C95E76;
END_STRUCT
END_TYPE

// ---- DUTs/IO/Boxes/KL1408_8EF4D3E9.TcDUT
{attribute 'GeneratedUsingTerminal: KL1408'}
{attribute addProperty BoxType "KL1408"}
{attribute addProperty Description ""}
{attribute addProperty Physics ""}
{attribute addProperty Id "Channel_1AT %I*Channel_87C95E760Channel_2AT %I*Channel_87C95E760Channel_3AT %I*Channel_87C95E760Channel_4AT %I*Channel_87C95E760Channel_5AT %I*Channel_87C95E760Channel_6AT %I*Channel_87C95E760Channel_7AT %I*Channel_87C95E760Channel_8AT %I*Channel_87C95E760"}
{attribute addProperty CRC "2398409705"}
{attribute addProperty Size "0"}
TYPE KL1408_8EF4D3E9 :
STRUCT
	{attribute addProperty Name "Channel_1"}
	Channel_1 : Channel_87C95E76;
	{attribute addProperty Name "Channel_2"}
	Channel_2 : Channel_87C95E76;
	{attribute addProperty Name "Channel_3"}
	Channel_3 : Channel_87C95E76;
	{attribute addProperty Name "Channel_4"}
	Channel_4 : Channel_87C95E76;
	{attribute addProperty Name "Channel_5"}
	Channel_5 : Channel_87C95E76;
	{attribute addProperty Name "Channel_6"}
	Channel_6 : Channel_87C95E76;
	{attribute addProperty Name "Channel_7"}
	Channel_7 : Channel_87C95E76;
	{attribute addProperty Name "Channel_8"}
	Channel_8 : Channel_87C95E76;
END_STRUCT
END_TYPE

// ---- DUTs/IO/Boxes/KL1412_BB38DA8F.TcDUT
{attribute 'GeneratedUsingTerminal: KL1412'}
{attribute addProperty BoxType "KL1412"}
{attribute addProperty Description ""}
{attribute addProperty Physics ""}
{attribute addProperty Id "Channel_1AT %I*Channel_87C95E760Channel_2AT %I*Channel_87C95E760"}
{attribute addProperty CRC "3141065359"}
{attribute addProperty Size "0"}
TYPE KL1412_BB38DA8F :
STRUCT
	{attribute addProperty Name "Channel_1"}
	Channel_1 : Channel_87C95E76;
	{attribute addProperty Name "Channel_2"}
	Channel_2 : Channel_87C95E76;
END_STRUCT
END_TYPE

// ---- DUTs/IO/Boxes/KL1414_4A257D2B.TcDUT
{attribute 'GeneratedUsingTerminal: KL1414'}
{attribute addProperty BoxType "KL1414"}
{attribute addProperty Description ""}
{attribute addProperty Physics ""}
{attribute addProperty Id "Channel_1AT %I*Channel_87C95E760Channel_2AT %I*Channel_87C95E760Channel_3AT %I*Channel_87C95E760Channel_4AT %I*Channel_87C95E760"}
{attribute addProperty CRC "1243970859"}
{attribute addProperty Size "0"}
TYPE KL1414_4A257D2B :
STRUCT
	{attribute addProperty Name "Channel_1"}
	Channel_1 : Channel_87C95E76;
	{attribute addProperty Name "Channel_2"}
	Channel_2 : Channel_87C95E76;
	{attribute addProperty Name "Channel_3"}
	Channel_3 : Channel_87C95E76;
	{attribute addProperty Name "Channel_4"}
	Channel_4 : Channel_87C95E76;
END_STRUCT
END_TYPE

// ---- DUTs/IO/Boxes/KL1418_8EF4D3E9.TcDUT
{attribute 'GeneratedUsingTerminal: KL1418'}
{attribute addProperty BoxType "KL1418"}
{attribute addProperty Description ""}
{attribute addProperty Physics ""}
{attribute addProperty Id "Channel_1AT %I*Channel_87C95E760Channel_2AT %I*Channel_87C95E760Channel_3AT %I*Channel_87C95E760Channel_4AT %I*Channel_87C95E760Channel_5AT %I*Channel_87C95E760Channel_6AT %I*Channel_87C95E760Channel_7AT %I*Channel_87C95E760Channel_8AT %I*Channel_87C95E760"}
{attribute addProperty CRC "2398409705"}
{attribute addProperty Size "0"}
TYPE KL1418_8EF4D3E9 :
STRUCT
	{attribute addProperty Name "Channel_1"}
	Channel_1 : Channel_87C95E76;
	{attribute addProperty Name "Channel_2"}
	Channel_2 : Channel_87C95E76;
	{attribute addProperty Name "Channel_3"}
	Channel_3 : Channel_87C95E76;
	{attribute addProperty Name "Channel_4"}
	Channel_4 : Channel_87C95E76;
	{attribute addProperty Name "Channel_5"}
	Channel_5 : Channel_87C95E76;
	{attribute addProperty Name "Channel_6"}
	Channel_6 : Channel_87C95E76;
	{attribute addProperty Name "Channel_7"}
	Channel_7 : Channel_87C95E76;
	{attribute addProperty Name "Channel_8"}
	Channel_8 : Channel_87C95E76;
END_STRUCT
END_TYPE

// ---- DUTs/IO/Boxes/KL1434_4A257D2B.TcDUT
{attribute 'GeneratedUsingTerminal: KL1434'}
{attribute addProperty BoxType "KL1434"}
{attribute addProperty Description ""}
{attribute addProperty Physics ""}
{attribute addProperty Id "Channel_1AT %I*Channel_87C95E760Channel_2AT %I*Channel_87C95E760Channel_3AT %I*Channel_87C95E760Channel_4AT %I*Channel_87C95E760"}
{attribute addProperty CRC "1243970859"}
{attribute addProperty Size "0"}
TYPE KL1434_4A257D2B :
STRUCT
	{attribute addProperty Name "Channel_1"}
	Channel_1 : Channel_87C95E76;
	{attribute addProperty Name "Channel_2"}
	Channel_2 : Channel_87C95E76;
	{attribute addProperty Name "Channel_3"}
	Channel_3 : Channel_87C95E76;
	{attribute addProperty Name "Channel_4"}
	Channel_4 : Channel_87C95E76;
END_STRUCT
END_TYPE

// ---- DUTs/IO/Boxes/KL1488_8EF4D3E9.TcDUT
{attribute 'GeneratedUsingTerminal: KL1488'}
{attribute addProperty BoxType "KL1488"}
{attribute addProperty Description ""}
{attribute addProperty Physics ""}
{attribute addProperty Id "Channel_1AT %I*Channel_87C95E760Channel_2AT %I*Channel_87C95E760Channel_3AT %I*Channel_87C95E760Channel_4AT %I*Channel_87C95E760Channel_5AT %I*Channel_87C95E760Channel_6AT %I*Channel_87C95E760Channel_7AT %I*Channel_87C95E760Channel_8AT %I*Channel_87C95E760"}
{attribute addProperty CRC "2398409705"}
{attribute addProperty Size "0"}
TYPE KL1488_8EF4D3E9 :
STRUCT
	{attribute addProperty Name "Channel_1"}
	Channel_1 : Channel_87C95E76;
	{attribute addProperty Name "Channel_2"}
	Channel_2 : Channel_87C95E76;
	{attribute addProperty Name "Channel_3"}
	Channel_3 : Channel_87C95E76;
	{attribute addProperty Name "Channel_4"}
	Channel_4 : Channel_87C95E76;
	{attribute addProperty Name "Channel_5"}
	Channel_5 : Channel_87C95E76;
	{attribute addProperty Name "Channel_6"}
	Channel_6 : Channel_87C95E76;
	{attribute addProperty Name "Channel_7"}
	Channel_7 : Channel_87C95E76;
	{attribute addProperty Name "Channel_8"}
	Channel_8 : Channel_87C95E76;
END_STRUCT
END_TYPE

// ---- DUTs/IO/Boxes/KL1498_8EF4D3E9.TcDUT
{attribute 'GeneratedUsingTerminal: KL1498'}
{attribute addProperty BoxType "KL1498"}
{attribute addProperty Description ""}
{attribute addProperty Physics ""}
{attribute addProperty Id "Channel_1AT %I*Channel_87C95E760Channel_2AT %I*Channel_87C95E760Channel_3AT %I*Channel_87C95E760Channel_4AT %I*Channel_87C95E760Channel_5AT %I*Channel_87C95E760Channel_6AT %I*Channel_87C95E760Channel_7AT %I*Channel_87C95E760Channel_8AT %I*Channel_87C95E760"}
{attribute addProperty CRC "2398409705"}
{attribute addProperty Size "0"}
TYPE KL1498_8EF4D3E9 :
STRUCT
	{attribute addProperty Name "Channel_1"}
	Channel_1 : Channel_87C95E76;
	{attribute addProperty Name "Channel_2"}
	Channel_2 : Channel_87C95E76;
	{attribute addProperty Name "Channel_3"}
	Channel_3 : Channel_87C95E76;
	{attribute addProperty Name "Channel_4"}
	Channel_4 : Channel_87C95E76;
	{attribute addProperty Name "Channel_5"}
	Channel_5 : Channel_87C95E76;
	{attribute addProperty Name "Channel_6"}
	Channel_6 : Channel_87C95E76;
	{attribute addProperty Name "Channel_7"}
	Channel_7 : Channel_87C95E76;
	{attribute addProperty Name "Channel_8"}
	Channel_8 : Channel_87C95E76;
END_STRUCT
END_TYPE

// ---- DUTs/IO/Boxes/KL1501_EE1D4506.TcDUT
{attribute 'GeneratedUsingTerminal: KL1501'}
{attribute addProperty BoxType "KL1501"}
{attribute addProperty Description ""}
{attribute addProperty Physics ""}
{attribute addProperty Id "Channel_1AT %Q*Channel_3C1A65000"}
{attribute addProperty CRC "3994895622"}
{attribute addProperty Size "0"}
TYPE KL1501_EE1D4506 :
STRUCT
	{attribute addProperty Name "Channel_1"}
	Channel_1 : Channel_3C1A6500;
END_STRUCT
END_TYPE

// ---- DUTs/IO/Boxes/KL_62DC61BC.TcDUT
{attribute 'GeneratedUsingTerminal: KL1501-0001'}
{attribute addProperty BoxType "KL1501-0001"}
{attribute addProperty Description ""}
{attribute addProperty Physics ""}
{attribute addProperty Id "Channel_1AT %Q*Channel_B5275D8E0"}
{attribute addProperty CRC "1658610108"}
{attribute addProperty Size "0"}
TYPE KL_62DC61BC :
STRUCT
	{attribute addProperty Name "Channel_1"}
	Channel_1 : Channel_B5275D8E;
END_STRUCT
END_TYPE

// ---- DUTs/IO/Boxes/KL1512_78388DBB.TcDUT
{attribute 'GeneratedUsingTerminal: KL1512'}
{attribute addProperty BoxType "KL1512"}
{attribute addProperty Description ""}
{attribute addProperty Physics ""}
{attribute addProperty Id "Channel_1AT %Q*Channel_03CEAA5E0Channel_2AT %Q*Channel_03CEAA5E0"}
{attribute addProperty CRC "2016972219"}
{attribute addProperty Size "0"}
TYPE KL1512_78388DBB :
STRUCT
	{attribute addProperty Name "Channel_1"}
	Channel_1 : Channel_03CEAA5E;
	{attribute addProperty Name "Channel_2"}
	Channel_2 : Channel_03CEAA5E;
END_STRUCT
END_TYPE

// ---- DUTs/IO/Boxes/KL1702_BB38DA8F.TcDUT
{attribute 'GeneratedUsingTerminal: KL1702'}
{attribute addProperty BoxType "KL1702"}
{attribute addProperty Description ""}
{attribute addProperty Physics ""}
{attribute addProperty Id "Channel_1AT %I*Channel_87C95E760Channel_2AT %I*Channel_87C95E760"}
{attribute addProperty CRC "3141065359"}
{attribute addProperty Size "0"}
TYPE KL1702_BB38DA8F :
STRUCT
	{attribute addProperty Name "Channel_1"}
	Channel_1 : Channel_87C95E76;
	{attribute addProperty Name "Channel_2"}
	Channel_2 : Channel_87C95E76;
END_STRUCT
END_TYPE

// ---- DUTs/IO/Boxes/KL1704_4A257D2B.TcDUT
{attribute 'GeneratedUsingTerminal: KL1704'}
{attribute addProperty BoxType "KL1704"}
{attribute addProperty Description ""}
{attribute addProperty Physics ""}
{attribute addProperty Id "Channel_1AT %I*Channel_87C95E760Channel_2AT %I*Channel_87C95E760Channel_3AT %I*Channel_87C95E760Channel_4AT %I*Channel_87C95E760"}
{attribute addProperty CRC "1243970859"}
{attribute addProperty Size "0"}
TYPE KL1704_4A257D2B :
STRUCT
	{attribute addProperty Name "Channel_1"}
	Channel_1 : Channel_87C95E76;
	{attribute addProperty Name "Channel_2"}
	Channel_2 : Channel_87C95E76;
	{attribute addProperty Name "Channel_3"}
	Channel_3 : Channel_87C95E76;
	{attribute addProperty Name "Channel_4"}
	Channel_4 : Channel_87C95E76;
END_STRUCT
END_TYPE

// ---- DUTs/IO/Boxes/KL1712_BB38DA8F.TcDUT
{attribute 'GeneratedUsingTerminal: KL1712'}
{attribute addProperty BoxType "KL1712"}
{attribute addProperty Description ""}
{attribute addProperty Physics ""}
{attribute addProperty Id "Channel_1AT %I*Channel_87C95E760Channel_2AT %I*Channel_87C95E760"}
{attribute addProperty CRC "3141065359"}
{attribute addProperty Size "0"}
TYPE KL1712_BB38DA8F :
STRUCT
	{attribute addProperty Name "Channel_1"}
	Channel_1 : Channel_87C95E76;
	{attribute addProperty Name "Channel_2"}
	Channel_2 : Channel_87C95E76;
END_STRUCT
END_TYPE

// ---- DUTs/IO/Boxes/KL_BB38DA8F.TcDUT
{attribute 'GeneratedUsingTerminal: KL1712-0001'}
{attribute addProperty BoxType "KL1712-0001"}
{attribute addProperty Description ""}
{attribute addProperty Physics ""}
{attribute addProperty Id "Channel_1AT %I*Channel_87C95E760Channel_2AT %I*Channel_87C95E760"}
{attribute addProperty CRC "3141065359"}
{attribute addProperty Size "0"}
TYPE KL_BB38DA8F :
STRUCT
	{attribute addProperty Name "Channel_1"}
	Channel_1 : Channel_87C95E76;
	{attribute addProperty Name "Channel_2"}
	Channel_2 : Channel_87C95E76;
END_STRUCT
END_TYPE

// ---- DUTs/IO/Boxes/KL1722_BB38DA8F.TcDUT
{attribute 'GeneratedUsingTerminal: KL1722'}
{attribute addProperty BoxType "KL1722"}
{attribute addProperty Description ""}
{attribute addProperty Physics ""}
{attribute addProperty Id "Channel_1AT %I*Channel_87C95E760Channel_2AT %I*Channel_87C95E760"}
{attribute addProperty CRC "3141065359"}
{attribute addProperty Size "0"}
TYPE KL1722_BB38DA8F :
STRUCT
	{attribute addProperty Name "Channel_1"}
	Channel_1 : Channel_87C95E76;
	{attribute addProperty Name "Channel_2"}
	Channel_2 : Channel_87C95E76;
END_STRUCT
END_TYPE

// ---- DUTs/IO/Boxes/KL1804_4A257D2B.TcDUT
{attribute 'GeneratedUsingTerminal: KL1804'}
{attribute addProperty BoxType "KL1804"}
{attribute addProperty Description ""}
{attribute addProperty Physics ""}
{attribute addProperty Id "Channel_1AT %I*Channel_87C95E760Channel_2AT %I*Channel_87C95E760Channel_3AT %I*Channel_87C95E760Channel_4AT %I*Channel_87C95E760"}
{attribute addProperty CRC "1243970859"}
{attribute addProperty Size "0"}
TYPE KL1804_4A257D2B :
STRUCT
	{attribute addProperty Name "Channel_1"}
	Channel_1 : Channel_87C95E76;
	{attribute addProperty Name "Channel_2"}
	Channel_2 : Channel_87C95E76;
	{attribute addProperty Name "Channel_3"}
	Channel_3 : Channel_87C95E76;
	{attribute addProperty Name "Channel_4"}
	Channel_4 : Channel_87C95E76;
END_STRUCT
END_TYPE

// ---- DUTs/IO/Boxes/KL1808_8EF4D3E9.TcDUT
{attribute 'GeneratedUsingTerminal: KL1808'}
{attribute addProperty BoxType "KL1808"}
{attribute addProperty Description ""}
{attribute addProperty Physics ""}
{attribute addProperty Id "Channel_1AT %I*Channel_87C95E760Channel_2AT %I*Channel_87C95E760Channel_3AT %I*Channel_87C95E760Channel_4AT %I*Channel_87C95E760Channel_5AT %I*Channel_87C95E760Channel_6AT %I*Channel_87C95E760Channel_7AT %I*Channel_87C95E760Channel_8AT %I*Channel_87C95E760"}
{attribute addProperty CRC "2398409705"}
{attribute addProperty Size "0"}
TYPE KL1808_8EF4D3E9 :
STRUCT
	{attribute addProperty Name "Channel_1"}
	Channel_1 : Channel_87C95E76;
	{attribute addProperty Name "Channel_2"}
	Channel_2 : Channel_87C95E76;
	{attribute addProperty Name "Channel_3"}
	Channel_3 : Channel_87C95E76;
	{attribute addProperty Name "Channel_4"}
	Channel_4 : Channel_87C95E76;
	{attribute addProperty Name "Channel_5"}
	Channel_5 : Channel_87C95E76;
	{attribute addProperty Name "Channel_6"}
	Channel_6 : Channel_87C95E76;
	{attribute addProperty Name "Channel_7"}
	Channel_7 : Channel_87C95E76;
	{attribute addProperty Name "Channel_8"}
	Channel_8 : Channel_87C95E76;
END_STRUCT
END_TYPE

// ---- DUTs/IO/Boxes/KL1809_65B88BEE.TcDUT
{attribute 'GeneratedUsingTerminal: KL1809'}
{attribute addProperty BoxType "KL1809"}
{attribute addProperty Description ""}
{attribute addProperty Physics ""}
{attribute addProperty Id "Channel_1AT %I*Channel_87C95E760Channel_2AT %I*Channel_87C95E760Channel_3AT %I*Channel_87C95E760Channel_4AT %I*Channel_87C95E760Channel_5AT %I*Channel_87C95E760Channel_6AT %I*Channel_87C95E760Channel_7AT %I*Channel_87C95E760Channel_8AT %I*Channel_87C95E760Channel_9AT %I*Channel_87C95E760Channel_10AT %I*Channel_87C95E760Channel_11AT %I*Channel_87C95E760Channel_12AT %I*Channel_87C95E760Channel_13AT %I*Channel_87C95E760Channel_14AT %I*Channel_87C95E760Channel_15AT %I*Channel_87C95E760Channel_16AT %I*Channel_87C95E760"}
{attribute addProperty CRC "1706593262"}
{attribute addProperty Size "0"}
TYPE KL1809_65B88BEE :
STRUCT
	{attribute addProperty Name "Channel_1"}
	Channel_1 : Channel_87C95E76;
	{attribute addProperty Name "Channel_2"}
	Channel_2 : Channel_87C95E76;
	{attribute addProperty Name "Channel_3"}
	Channel_3 : Channel_87C95E76;
	{attribute addProperty Name "Channel_4"}
	Channel_4 : Channel_87C95E76;
	{attribute addProperty Name "Channel_5"}
	Channel_5 : Channel_87C95E76;
	{attribute addProperty Name "Channel_6"}
	Channel_6 : Channel_87C95E76;
	{attribute addProperty Name "Channel_7"}
	Channel_7 : Channel_87C95E76;
	{attribute addProperty Name "Channel_8"}
	Channel_8 : Channel_87C95E76;
	{attribute addProperty Name "Channel_9"}
	Channel_9 : Channel_87C95E76;
	{attribute addProperty Name "Channel_10"}
	Channel_10 : Channel_87C95E76;
	{attribute addProperty Name "Channel_11"}
	Channel_11 : Channel_87C95E76;
	{attribute addProperty Name "Channel_12"}
	Channel_12 : Channel_87C95E76;
	{attribute addProperty Name "Channel_13"}
	Channel_13 : Channel_87C95E76;
	{attribute addProperty Name "Channel_14"}
	Channel_14 : Channel_87C95E76;
	{attribute addProperty Name "Channel_15"}
	Channel_15 : Channel_87C95E76;
	{attribute addProperty Name "Channel_16"}
	Channel_16 : Channel_87C95E76;
END_STRUCT
END_TYPE

// ---- DUTs/IO/Boxes/KL1814_4A257D2B.TcDUT
{attribute 'GeneratedUsingTerminal: KL1814'}
{attribute addProperty BoxType "KL1814"}
{attribute addProperty Description ""}
{attribute addProperty Physics ""}
{attribute addProperty Id "Channel_1AT %I*Channel_87C95E760Channel_2AT %I*Channel_87C95E760Channel_3AT %I*Channel_87C95E760Channel_4AT %I*Channel_87C95E760"}
{attribute addProperty CRC "1243970859"}
{attribute addProperty Size "0"}
TYPE KL1814_4A257D2B :
STRUCT
	{attribute addProperty Name "Channel_1"}
	Channel_1 : Channel_87C95E76;
	{attribute addProperty Name "Channel_2"}
	Channel_2 : Channel_87C95E76;
	{attribute addProperty Name "Channel_3"}
	Channel_3 : Channel_87C95E76;
	{attribute addProperty Name "Channel_4"}
	Channel_4 : Channel_87C95E76;
END_STRUCT
END_TYPE

// ---- DUTs/IO/Boxes/KL1819_65B88BEE.TcDUT
{attribute 'GeneratedUsingTerminal: KL1819'}
{attribute addProperty BoxType "KL1819"}
{attribute addProperty Description ""}
{attribute addProperty Physics ""}
{attribute addProperty Id "Channel_1AT %I*Channel_87C95E760Channel_2AT %I*Channel_87C95E760Channel_3AT %I*Channel_87C95E760Channel_4AT %I*Channel_87C95E760Channel_5AT %I*Channel_87C95E760Channel_6AT %I*Channel_87C95E760Channel_7AT %I*Channel_87C95E760Channel_8AT %I*Channel_87C95E760Channel_9AT %I*Channel_87C95E760Channel_10AT %I*Channel_87C95E760Channel_11AT %I*Channel_87C95E760Channel_12AT %I*Channel_87C95E760Channel_13AT %I*Channel_87C95E760Channel_14AT %I*Channel_87C95E760Channel_15AT %I*Channel_87C95E760Channel_16AT %I*Channel_87C95E760"}
{attribute addProperty CRC "1706593262"}
{attribute addProperty Size "0"}
TYPE KL1819_65B88BEE :
STRUCT
	{attribute addProperty Name "Channel_1"}
	Channel_1 : Channel_87C95E76;
	{attribute addProperty Name "Channel_2"}
	Channel_2 : Channel_87C95E76;
	{attribute addProperty Name "Channel_3"}
	Channel_3 : Channel_87C95E76;
	{attribute addProperty Name "Channel_4"}
	Channel_4 : Channel_87C95E76;
	{attribute addProperty Name "Channel_5"}
	Channel_5 : Channel_87C95E76;
	{attribute addProperty Name "Channel_6"}
	Channel_6 : Channel_87C95E76;
	{attribute addProperty Name "Channel_7"}
	Channel_7 : Channel_87C95E76;
	{attribute addProperty Name "Channel_8"}
	Channel_8 : Channel_87C95E76;
	{attribute addProperty Name "Channel_9"}
	Channel_9 : Channel_87C95E76;
	{attribute addProperty Name "Channel_10"}
	Channel_10 : Channel_87C95E76;
	{attribute addProperty Name "Channel_11"}
	Channel_11 : Channel_87C95E76;
	{attribute addProperty Name "Channel_12"}
	Channel_12 : Channel_87C95E76;
	{attribute addProperty Name "Channel_13"}
	Channel_13 : Channel_87C95E76;
	{attribute addProperty Name "Channel_14"}
	Channel_14 : Channel_87C95E76;
	{attribute addProperty Name "Channel_15"}
	Channel_15 : Channel_87C95E76;
	{attribute addProperty Name "Channel_16"}
	Channel_16 : Channel_87C95E76;
END_STRUCT
END_TYPE

// ---- DUTs/IO/Boxes/KL1859_C5B2A062.TcDUT
{attribute 'GeneratedUsingTerminal: KL1859'}
{attribute addProperty BoxType "KL1859"}
{attribute addProperty Description ""}
{attribute addProperty Physics ""}
{attribute addProperty Id "Channel_1AT %Q*Channel_70C997F30Channel_2AT %Q*Channel_70C997F30Channel_3AT %Q*Channel_70C997F30Channel_4AT %Q*Channel_70C997F30Channel_5AT %Q*Channel_70C997F30Channel_6AT %Q*Channel_70C997F30Channel_7AT %Q*Channel_70C997F30Channel_8AT %Q*Channel_70C997F30"}
{attribute addProperty CRC "3316818018"}
{attribute addProperty Size "0"}
TYPE KL1859_C5B2A062 :
STRUCT
	{attribute addProperty Name "Channel_1"}
	Channel_1 : Channel_70C997F3;
	{attribute addProperty Name "Channel_2"}
	Channel_2 : Channel_70C997F3;
	{attribute addProperty Name "Channel_3"}
	Channel_3 : Channel_70C997F3;
	{attribute addProperty Name "Channel_4"}
	Channel_4 : Channel_70C997F3;
	{attribute addProperty Name "Channel_5"}
	Channel_5 : Channel_70C997F3;
	{attribute addProperty Name "Channel_6"}
	Channel_6 : Channel_70C997F3;
	{attribute addProperty Name "Channel_7"}
	Channel_7 : Channel_70C997F3;
	{attribute addProperty Name "Channel_8"}
	Channel_8 : Channel_70C997F3;
END_STRUCT
END_TYPE

// ---- DUTs/IO/Boxes/KL1862_65B88BEE.TcDUT
{attribute 'GeneratedUsingTerminal: KL1862'}
{attribute addProperty BoxType "KL1862"}
{attribute addProperty Description ""}
{attribute addProperty Physics ""}
{attribute addProperty Id "Channel_1AT %I*Channel_87C95E760Channel_2AT %I*Channel_87C95E760Channel_3AT %I*Channel_87C95E760Channel_4AT %I*Channel_87C95E760Channel_5AT %I*Channel_87C95E760Channel_6AT %I*Channel_87C95E760Channel_7AT %I*Channel_87C95E760Channel_8AT %I*Channel_87C95E760Channel_9AT %I*Channel_87C95E760Channel_10AT %I*Channel_87C95E760Channel_11AT %I*Channel_87C95E760Channel_12AT %I*Channel_87C95E760Channel_13AT %I*Channel_87C95E760Channel_14AT %I*Channel_87C95E760Channel_15AT %I*Channel_87C95E760Channel_16AT %I*Channel_87C95E760"}
{attribute addProperty CRC "1706593262"}
{attribute addProperty Size "0"}
TYPE KL1862_65B88BEE :
STRUCT
	{attribute addProperty Name "Channel_1"}
	Channel_1 : Channel_87C95E76;
	{attribute addProperty Name "Channel_2"}
	Channel_2 : Channel_87C95E76;
	{attribute addProperty Name "Channel_3"}
	Channel_3 : Channel_87C95E76;
	{attribute addProperty Name "Channel_4"}
	Channel_4 : Channel_87C95E76;
	{attribute addProperty Name "Channel_5"}
	Channel_5 : Channel_87C95E76;
	{attribute addProperty Name "Channel_6"}
	Channel_6 : Channel_87C95E76;
	{attribute addProperty Name "Channel_7"}
	Channel_7 : Channel_87C95E76;
	{attribute addProperty Name "Channel_8"}
	Channel_8 : Channel_87C95E76;
	{attribute addProperty Name "Channel_9"}
	Channel_9 : Channel_87C95E76;
	{attribute addProperty Name "Channel_10"}
	Channel_10 : Channel_87C95E76;
	{attribute addProperty Name "Channel_11"}
	Channel_11 : Channel_87C95E76;
	{attribute addProperty Name "Channel_12"}
	Channel_12 : Channel_87C95E76;
	{attribute addProperty Name "Channel_13"}
	Channel_13 : Channel_87C95E76;
	{attribute addProperty Name "Channel_14"}
	Channel_14 : Channel_87C95E76;
	{attribute addProperty Name "Channel_15"}
	Channel_15 : Channel_87C95E76;
	{attribute addProperty Name "Channel_16"}
	Channel_16 : Channel_87C95E76;
END_STRUCT
END_TYPE

